// TwinCAT 3 PLC project MONETRuntime
// ProgramVersion: 3.1.4023.0
// libraries:
//   AstroBROT, * (BROT)
//   BROTLib, * (BROT)
//   Tc2_DataExchange, * (Beckhoff Automation GmbH)
//   Tc2_Math, * (Beckhoff Automation GmbH)
//   Tc2_MC2, * (Beckhoff Automation GmbH)
//   Tc2_MC2_Drive, * (Beckhoff Automation GmbH)
//   Tc2_NC, * (Beckhoff Automation GmbH)
//   Tc2_Standard, * (Beckhoff Automation GmbH)
//   Tc2_System, * (Beckhoff Automation GmbH)
//   Tc2_Utilities, * (Beckhoff Automation GmbH)
//   Tc3_IotBase, * (Beckhoff Automation GmbH)
//   Tc3_Module, * (Beckhoff Automation GmbH)
//   VisuDialogs, * (System)
//   VisuSymbols,3.5.10.0,System
// project tree:
//   DUTs/ E_Blink.TcDUT (not stored), E_Horn.TcDUT (not stored), E_TCSCommand.TcDUT (not stored), E_TCSErrors.TcDUT (not stored), E_TelescopeMode.TcDUT (not stored)
//   / GlobalTextList.TcGTLO, PlcTask.TcTTO (not stored), Visualization Manager.TcVMO (not stored)
//   GVLs/ GVL_Hydraulics.TcGVL (not stored), GVL_Main.TcGVL, GVL_pendant_control.TcGVL (not stored), GVL_Roof.TcGVL (not stored), GVL_Safety.TcGVL, GVL_Telescope.TcGVL
//   POUs/ AzimuthElevationControl.TcPOU, CoverControl.TcPOU, DerotatorControl.TcPOU, ElevationControl.TcPOU, FocusControl.TcPOU, HydraulicsControl.TcPOU, MAIN.TcPOU, PendantControl.TcPOU, RoofControl.TcPOU, PowerMonitoring.TcPOU, SafetyHandling.TcPOU, TelescopeAuxiliary.TcPOU, TelescopeControl.TcPOU
//   POUs/FunctionBlocks/ FB_AstroClock.TcPOU (not stored), FB_BLINK.TcPOU (not stored), FB_ButtonEnable.TcPOU (not stored), FB_Cover.TcPOU (not stored), FB_EventLog.TcPOU (not stored), FB_Horn.TcPOU (not stored), FB_LightTimer.TcPOU (not stored), FB_RFTRIG.TcPOU (not stored), FB_TimeAverage.TcPOU (not stored), FB_Timer.TcPOU (not stored), FB_TONTP.TcPOU (not stored), TelescopeAxisClass.TcPOU (not stored)
//   POUs/Functions/ CT2LST.TcPOU (not stored), F_Azimuthvelocity.TcPOU (not stored), F_DerotatorPosition2.TcPOU (not stored), F_Derotatorvelocity.TcPOU (not stored), F_Elevationvelocity.TcPOU (not stored), F_YREAL.TcPOU (not stored), NCError_TO_STRING.TcPOU (not stored), PointingModelAzimuth.TcPOU (not stored), PointingModelElevation.TcPOU (not stored), Refraction.TcPOU (not stored)
//   VISUs/ Hydraulics.TcVIS, Safety.TcVIS, Visualization.TcVIS

// ---- GVLs/GVL_Main.TcGVL
{attribute 'qualified_only'}
//TODO update to current RoboTel IOs
VAR_GLOBAL
	//DIN1 0.0
	//phase_available		AT%I*: BOOL;
	//not implemented on RoboTel
	//key_switch			AT%I*: BOOL;
	//DIN3 0.2
	key_switch_remote	AT%I*: BOOL;
	//DIN4 0.3
	start_switch		AT%I*: BOOL;
	//DIN5 0.4
	stop_switch			AT%I*: BOOL;
	//DIN8 0.7
	reset_switch		AT%I*: BOOL;
	
	//BT1
	main_cabinet_temperature	AT%I*: INT;
	//DIN15 1.6
	brake_clearing		AT%I*: BOOL;
	
	//DOUT1 0.0
	lamp_power			AT%Q*: BOOL;
	//DOUT2 0.1
	lamp_on_manual			AT%Q*: BOOL;
	//DOUT3 0.2
	lamp_error			AT%Q*: BOOL;
	
	(*
	NeutralCurrentGuardWarning		AT%I*:	BOOL;
	NeutralCurrentGuarError			AT%I*:	BOOL;
	ActivePowerGuardWarning			AT%I*:	BOOL;
	ActivePowerGuardError			AT%I*:	BOOL;
	ApparentPowerGuardWarning		AT%I*:	BOOL;
	ApparentPowerGuardError			AT%I*:	BOOL;
	*)
	//ActivePower						AT%I*:	REAL;
	//ActiveEnergy					AT%I*:	LINT;
	//NeutralLineCurrent				AT%I*:	REAL;
END_VAR

// ---- GVLs/GVL_Safety.TcGVL
{attribute 'qualified_only'}
VAR_GLOBAL
	// Safety Error Condition
	Error		AT%I*:	BOOL;
	// Run/Stop Safety
	Run			AT%Q*:	BOOL;
	// Restart Safety
	Restart		AT%Q*:	BOOL;
	// Error Acknowledgement 
	ErrAck		AT%Q*:	BOOL;
	// Stop signal coming from Safety
	// Stop		AT%I*:	BOOL;
	
	Reset_STO_Azimuth		AT%Q*: BOOL;
	Reset_STO_Elevation		AT%Q*: BOOL;
	Reset_STO_Derotator		AT%Q*: BOOL;
END_VAR

// ---- GVLs/GVL_Telescope.TcGVL
{attribute 'qualified_only'}
VAR_GLOBAL
	// DIN28 3.3 (absolute)
	azimut_limit_switch	AT%I*: BOOL;

	//Horn 4.7
	horn			AT%Q*: BOOL;
	
END_VAR

// ---- POUs/AzimuthElevationControl.TcPOU
PROGRAM AzimuthElevationControl
VAR_INPUT
	// enable the axis and its position control loop
	Enable:		BOOL;
	// reset the axis
	Reset: 		BOOL;
	// decrease azimuth
	left:		BOOL;
	// increase azimuth
	right: 		BOOL;
	// Move azimuth to given position
	MoveAxis:	BOOL;
	// Home the axis
	HomeAxis:	BOOL;
	// enable tracking
	Tracking:	BOOL;
	// position to move the axis to
	position: 	LREAL;
	// set the Velocity of the axis
	velocity:	LREAL;
	// stop the Axis
	StopAxis:	BOOL;
	// diagnostic reset
	bSoEReset:	BOOL;
	comm: I_Comm;
END_VAR
VAR_IN_OUT
	HydraulicsControl : FB_HydraulicsControl;
END_VAR
VAR_OUTPUT
	// error state of the axis
	error: 			BOOL;
	// error ID of the axis
	ErrorID:		UDINT;
	// actual_position of the axis
	act_position:	LREAL;
	// is the axis calibrated
	calibrated:		BOOL;
	// drive is ready
	ready:			BOOL;
	// time to reach target position
	slewtime:		LREAL;
END_VAR
VAR
	AzimuthAxis:		FB_Axis2;
	AzimuthCalibration: MC_SetPosition;
	//fbSoEReset:			FB_SoEReset;
	AzimuthAxisEvent: 	FB_EventLog;
	AzimuthDiagnosticEvent: 	FB_EventLog;
	// delay until commutator angle is measured
	readydelay:			TON;
	HomeDelay:			FB_TONTP;
	TorqueError:		TON := (PT := T#3S);
	azimuth_torque: 	REAL;
	TorqueWarning:		FB_EventLog;
	CalibrationEvent:	FB_Eventlog;
	ReadParameter:		MC_ReadParameter;
	getlastposition:	BOOL := TRUE;
	azimuth_rest_timer:	TON;
	azimuth_at_rest:	BOOL;
	fbSoEReset: 		FB_SoEReset;
	DiagnosticError:	BOOL;
END_VAR
VAR CONSTANT
	// reference position for homing
	// homing_position:		LREAL := 439.0; // was 442 - -21.21 = 463.21; 463 + 24 = 439
	// current position of the calibration cam encoder zero index. Apply an offset here if necessary
	calibration_position:	LREAL :=  212.75; //208.4983;//208.6273; //208.6073; // 208.7122869;//207.0092; // 208.2342; 
END_VAR
VAR PERSISTENT
	last_position:	LREAL := -1.0;
END_VAR

(* Azimuth Axis control section
Power must be on and brake must be open for the axis to operate
*)

// generate the ready signal after enabling the drive
readydelay(IN :=  AzimuthAxis.Enable, PT := T#3000MS, Q=> ready);

// limit the input position angle
position := LIMIT(0.0, position, 450.0);

// conduct the calibrated signal
calibrated := AzimuthAxis.Calibrated;

IF Calibrated OR Error THEN
	HomeAxis := FALSE;
	getlastposition := FALSE;
END_IF
	
IF HomeAxis THEN
	position := calibration_position;
END_IF

IF HomeDelay.Q THEN
	position := calibration_position;
	MoveAxis := TRUE;
END_IF

// perform a recalibration on the last known position
AzimuthCalibration(
	Axis := GVL_Telescope.AzimuthAxisRef,
	Execute := getlastposition AND last_position>=0.0 AND NOT Calibrated,
	Position := last_position);

IF AzimuthCalibration.Done THEN
	getlastposition := FALSE;
END_IF

IF Calibrated THEN
	last_position := act_position;
END_IF

// enable the azimuth if not moved by the power chain. Sorry for the hack
azimuth_rest_timer(IN := HydraulicsControl.brake_open AND 
				(ABS(GVL_Telescope.AzimuthAxisRef.NcToPlc.ActVelo) < 0.01), PT := T#2S);
// if azimuth at rest or calibrated, allow enabling the azimuth
IF azimuth_rest_timer.Q or calibrated THEN
	azimuth_at_rest := TRUE;
ELSIF HydraulicsControl.brake_closed THEN
	azimuth_at_rest := FALSE;
END_IF
	
// deactivate limit switches on homing
MC_SetAcceptBlockedDriveSignal(
	Axis := GVL_Telescope.AzimuthAxisRef, 
	Enable := HomeAxis);

AzimuthAxis(	
	Enable := 			enable AND azimuth_at_rest AND NOT GVL_Telescope.azimut_limit_switch,
	Reset := 			reset,
	MoveAxis :=			MoveAxis,
	HomeAxis := 		HomeAxis,
	StopAxis :=			StopAxis,
	Tracking :=			Tracking,
	Position := 		position, 
	Velocity :=			velocity,
	Enable_Positive := 	GVL_Telescope.Azimuth_inputs.1 OR HomeAxis,
	Enable_Negative := 	GVL_Telescope.Azimuth_inputs.0,
	Jog_Forward :=		right,
	Jog_Backwards := 	left,
	bCalibrationCam :=	NOT GVL_Telescope.Azimuth_inputs.1,
	ActualPosition => 	act_position,
	Error => 			error,
	ErrorID => 			ErrorID,
	AxisRef :=			GVL_Telescope.AzimuthAxisRef);

IF bSoEReset THEN
	last_position := -1.0;
	fbSoEReset(
		Axis := GVL_Telescope.AzimuthAxisRef,
		Execute := TRUE,
		Timeout := DEFAULT_ADS_TIMEOUT);
 	IF fbSoEReset.Busy THEN
		fbSoEReset(Axis := GVL_Telescope.AzimuthAxisRef, Execute := FALSE);
	ELSE
		bSoEReset := FALSE;
		Reset := TRUE;
	END_IF
END_IF 

IF AzimuthAxis.MoveDone THEN
	MoveAxis := FALSE;
END_IF

IF AzimuthAxis.HomeDone THEN
	HomeAxis := FALSE;
END_IF
	
IF AzimuthAxis.ResetDone THEN
	reset := FALSE;
END_IF

IF AzimuthAxis.StopDone THEN
	StopAxis := FALSE;
END_IF
DiagnosticError := FALSE;
IF GVL_Telescope.Azimuth_diagnostic < 16#D012 AND GVL_Telescope.Azimuth_diagnostic > 16#D014 THEN
	DiagnosticError :=TRUE;
	ErrorID := GVL_Telescope.Azimuth_diagnostic;
END_IF

ReadParameter(	Axis := GVL_Telescope.AzimuthAxisRef, Enable := AzimuthAxis.InMotion, 
				ParameterNumber := MC_AxisParameter.AxisRemainingTimeToGo, 
				ReadMode := E_ReadMode.READMODE_CYCLIC);
IF ReadParameter.Valid THEN
	slewtime := ReadParameter.Value;
END_IF

azimuth_torque := GVL_Telescope.Azimuth_torque / 10.0;
TorqueError(IN := ABS(azimuth_torque) > 50.0);


AzimuthAxisEvent(	
	Trigger := 		Error, 
	Level := 		ADSLOG_MSGTYPE_ERROR,
	FormatString :=	'Azimuth Axis Error: %s',
	OnMessage := 	NCError_TO_STRING(ErrorID),
	Comm := comm);
	
AzimuthDiagnosticEvent(	
	Trigger := 		DiagnosticError,
	Level := 		ADSLOG_MSGTYPE_ERROR,
	FormatString :=	'Azimuth Axis Diagnostic Error: %s',
	OnMessage := 	NCError_TO_STRING(GVL_Telescope.Azimuth_diagnostic),
	Comm := comm);
	
TorqueWarning(	
	Trigger := 		TorqueError.Q, 
	Level := 		ADSLOG_MSGTYPE_WARN,
	FormatString :=	'%s',
	OnMessage := 	'Azimuth torque is high.',
	Comm := comm);
	
CalibrationEvent(
	Trigger := 		Calibrated, 
	Level := 		ADSLOG_MSGTYPE_HINT,
	FormatString :=	'%s',
	OnMessage := 	'Azimuth axis is calibrated.',
	Comm := comm);

END_PROGRAM

// ---- POUs/HydraulicsControl.TcPOU
PROGRAM HydraulicsControl
VAR_INPUT
	// start the hydraulics
	enable:		BOOL := FALSE;
	// reset any hydraulics error
	reset: 		BOOL;
	// manual override to start the suction pump
	suction_manual:	BOOL;
	//manual override to stop the pump
	pump_manual_stop: BOOL;
END_VAR
VAR_OUTPUT
	// status of the brake: is the brake open?
	brake_open:			BOOL;
	// is the brake closed?
	brake_closed:		BOOL;
	// pump is running, but the pressure remains low
	pressure_failure:	BOOL;
	// suction was started, but it is not running
	suction_failure:	BOOL;
	// main pump is running but suction has a timeout
	hydraulics_failure:	BOOL;
	main_pump_failure: BOOL;
	// oil is low
	oil_low:			BOOL;
	// oil is high (unused?)
	oil_high:			BOOL;
	// oil pressure is 25 bars
	oil_pressure_OK:	BOOL;
	// oil is on reserve
	oil_warning:		BOOL;
	// oil filter is dirty
	oil_filter_dirty:	BOOL;
	// oil is below 10°C
	oil_cold:			BOOL;
	// oil is above 50°C
	oil_hot:			BOOL;
	// main pump is running
	pump_running:		BOOL;
	// suction pump is running
	suction_running :	BOOL := FALSE;
	// error condition
	error: 				BOOL;
END_VAR
VAR
	// command to open the brake
	iopen_brake:	BOOL := FALSE;
	// command to open the brake
	iclose_brake: BOOL;
	// monitors the pressure of the pump is running
	pressure_watchdog:	TON;
	// monitors the activation of the suction pump
	suction_watchdog: TON;
	// monitors the activation of the main pump
	main_pump_watchdog:	TON;
	// watch the hydraulics and suction pumps
	hydraulics_watchdog: TON;
	// represents the state of the main pump
	oil_pump_state:		RS;
	// represents the state of the brake
	brake_state: 		RS;
	// wait for the brake to open after pressure has been established
	brake_open_delay:	TON;
	// report brake opend after a short delay
	brake_opened_delay:	TON;
	// error state (set dominant)
	error_state:	SR;
	// trigger for suction pump
	suction_trigger:	SR;
	// timer to shut off hydraulics after break was closed
	hydraulics_off_timer:	TON  := (PT := T#300S);
	off_trigger:	F_TRIG;
	oil_level, last_oil_level:		REAL;
	HydraulicsLog,
	PumpLog,
	ReserveLog,
	oil_low_log,
	FilterLog,
	oil_max_log,
	OverTemperatureLog,
	UnderTemperatureLog,
	SuctionLog,
	HydraulicsFailureLog,
	BrakeClearingWarning,
	BrakeHydraulicsWarning,
	BrakeWarning: FB_EventLog;
	
	// measures the operating cycle of the suction pump
	StatusWord, LastStatus:	UDINT;
END_VAR

(* 
Main control Logic for the Hydraulics system
* power on delay for main pump and suction pump
* start main pump if main control is ready (button pressed or remote)
* start suction pump if maximum in pan is reached
* suction pump runs for 60 seconds
* stop main pump if oil is low
* stop main pump if pressure fails for 10 seconds
*)
oil_low := NOT GVL_Hydraulics.oil_low;
oil_high := NOT GVL_Hydraulics.oil_high;
oil_warning := GVL_Hydraulics.oil_reserve;
oil_pressure_OK := GVL_Hydraulics.oil_pressure_OK;
oil_filter_dirty := NOT GVL_Hydraulics.oilfilter_dirty;
oil_cold := NOT GVL_Hydraulics.oil_undertemperature;
oil_hot := GVL_Hydraulics.oil_overtemperature;
oil_level := F_YREAL(GVL_Hydraulics.oil_level, 0, 16383, 0.0, 5.0);
pump_running := GVL_Hydraulics.pump_running;
suction_running := GVL_Hydraulics.suction_running;

error_state(SET1 := pressure_failure OR	suction_failure OR hydraulics_failure OR oil_low OR main_pump_failure,
			RESET := reset,
			Q1 => error);
// clear reset, if no error present

IF NOT error THEN
	reset := FALSE;
END_IF

oil_pump_state(SET := enable,
				RESET1 := NOT enable OR error OR pump_manual_stop OR GVL_Hydraulics.oilpan_maximum);

GVL_Hydraulics.oil_pump_enable := oil_pump_state.Q1;

(* This section controls the hydraulic brake responsible for azimuth and elevation. 
Especially the elevation is imbalanced if not in the position control loop. 
The brake must only be opened, if the elevation drive is activated concurrently.
*)


// close the brake if the pump is not running	
IF iclose_brake OR NOT pump_running THEN 
	iopen_brake := FALSE;
END_IF

// wait for pressure to build up (hack for oil_pressure_ok)
brake_open_delay(IN := pump_running AND oil_pressure_OK,
				PT := T#3S);
		
brake_state(SET := brake_open_delay.Q AND iopen_brake AND MAIN.brake_clearing,
			RESET1 := GVL_Telescope.azimut_limit_switch 
					  OR iclose_brake 
					  OR NOT pump_running
					  OR NOT MAIN.brake_clearing,
			Q1 => GVL_Telescope.brake_azimuth_eve);

// signal that the brake is open after one second
brake_opened_delay(	IN :=brake_state.Q1, 
					PT := T#1000MS,
					Q => brake_open);

brake_closed := NOT brake_open;
IF brake_closed THEN
	iclose_brake := FALSE;
END_IF
// turn off the hydraulics if the brake is closed and the pump is still running
hydraulics_off_timer(IN := brake_closed AND enable );
off_trigger(CLK := hydraulics_off_timer.Q);

IF hydraulics_off_timer.Q THEN
	enable := FALSE;
END_IF

(* This is the end of the brake control section *)

suction_trigger(SET1 := GVL_Hydraulics.oilpan_maximum OR oil_level>2.9,
				RESET := oil_level<1.2);
GVL_Hydraulics.oil_suction_enable := suction_trigger.Q1 OR suction_manual;					
suction_watchdog(IN := GVL_Hydraulics.oil_suction_enable AND NOT suction_running,
					PT := T#15S,
					Q => suction_failure);
					
pressure_watchdog(IN := GVL_Hydraulics.oil_pump_enable AND 
						NOT oil_pressure_OK,
					PT := T#30S,
				  Q => pressure_failure);
hydraulics_watchdog(IN := pump_running AND NOT suction_running,
						PT := T#140S,
						Q => hydraulics_failure);

main_pump_watchdog(IN := GVL_Hydraulics.oil_pump_enable AND NOT pump_running,
					PT := T#10S,
					Q => main_pump_failure);

StatusWord.0 := oil_low;
StatusWord.1 := oil_high;
StatusWord.2 := oil_warning;
StatusWord.3 := oil_pressure_OK;
StatusWord.4 := oil_filter_dirty;
StatusWord.5 := oil_cold;
StatusWord.6 := oil_hot;
StatusWord.7 := brake_open;
StatusWord.8 := GVL_Main.brake_clearing;
StatusWord.9 := pump_running;
StatusWord.10 := suction_running;
StatusWord.11 := GVL_Hydraulics.oilpan_maximum;
StatusWord.12 := GVL_Hydraulics.oil_pump_enable;
StatusWord.13 := GVL_Hydraulics.oil_suction_enable;
IF ABS(last_oil_level - oil_level) > 0.02 THEN
	StatusWord.15 := TRUE;
	last_oil_level := oil_level;
ELSE
	StatusWord.15 := FALSE;
END_IF

IF StatusWord<>LastStatus THEN // publish new payload every second
	LastStatus := StatusWord;
	MAIN.MQTTClient.Publish('hydraulics', 'base', 'OilLow',			BOOL_TO_STRING(oil_low));
	MAIN.MQTTClient.Publish('hydraulics', 'base', 'OilHigh',		BOOL_TO_STRING(oil_high));
	MAIN.MQTTClient.Publish('hydraulics', 'base', 'OilMaximum',		BOOL_TO_STRING(GVL_Hydraulics.oilpan_maximum));
	MAIN.MQTTClient.Publish('hydraulics', 'base', 'OilReserve',		BOOL_TO_STRING(oil_warning));
	MAIN.MQTTClient.Publish('hydraulics', 'base', 'OilPressureOK', 	BOOL_TO_STRING(oil_pressure_OK));
	MAIN.MQTTClient.Publish('hydraulics', 'base', 'OilFilterDirty',	BOOL_TO_STRING(oil_filter_dirty));
	MAIN.MQTTClient.Publish('hydraulics', 'base', 'OilCold',		BOOL_TO_STRING(oil_cold));
	MAIN.MQTTClient.Publish('hydraulics', 'base', 'OilHot',			BOOL_TO_STRING(oil_Hot));
	MAIN.MQTTClient.Publish('hydraulics', 'base', 'BrakeOpen',		BOOL_TO_STRING(brake_open));
	MAIN.MQTTClient.Publish('hydraulics', 'base', 'BrakeClearing',	BOOL_TO_STRING(GVL_Main.brake_clearing));
	MAIN.MQTTClient.Publish('hydraulics', 'base', 'PumpRunning',	BOOL_TO_STRING(pump_running));
	MAIN.MQTTClient.Publish('hydraulics', 'base', 'SuctionRunning',	BOOL_TO_STRING(suction_running));
	MAIN.MQTTClient.Publish('hydraulics', 'base', 'OilLevel',		REAL_TO_STRING(oil_level));
	MAIN.MQTTClient.Publish('hydraulics', 'base', 'StatusWord',		UDINT_TO_STRING(StatusWord));
END_IF


				  				  
HydraulicsLog(Trigger := pressure_failure OR main_pump_failure,
				Level := ADSLOG_MSGTYPE_ERROR,
				FormatString := 'Main hydraulics pump / pressure: %s',
				OnMessage := 'FAILURE',
				OffMessage := 'OK',
				OffLevel := ADSLOG_MSGTYPE_HINT);

PumpLog(Trigger := pump_running,
				Level := ADSLOG_MSGTYPE_HINT,
				FormatString := 'Main hydraulics pump: %s',
				OnMessage := 'START',
				OffMessage := 'STOP',
				OffLevel := ADSLOG_MSGTYPE_HINT);
	
ReserveLog(Trigger := oil_warning,
			Level := ADSLOG_MSGTYPE_WARN,
			FormatString := 'oil reserve: %s',
			OnMessage := 'LOW',
			OffMessage := 'OK',
			OffLevel := ADSLOG_MSGTYPE_HINT);

oil_low_log(Trigger := oil_low,
				Level := ADSLOG_MSGTYPE_ERROR,
				FormatString := 'oil level: %s',
				OnMessage := 'LOW',
				OffMessage := 'OK',
				OffLevel := ADSLOG_MSGTYPE_HINT);

oil_max_log(Trigger := GVL_Hydraulics.oilpan_maximum,
				Level := ADSLOG_MSGTYPE_ERROR,
				FormatString := 'oil level: %s',
				OnMessage := 'MAXIMUM',
				OffMessage := 'OK',
				OffLevel := ADSLOG_MSGTYPE_HINT);	
				
FilterLog(Trigger := oil_filter_dirty,
				Level := ADSLOG_MSGTYPE_WARN,
				FormatString := 'Hydraulics Filter is %s',
				OnMessage := 'dirty.');

OverTemperatureLog(Trigger := oil_hot,
				Level := ADSLOG_MSGTYPE_WARN,
				FormatString := 'Hydraulics Temperature is %s',
				OnMessage := 'high.');
				
UnderTemperatureLog(Trigger := oil_cold,
				Level := ADSLOG_MSGTYPE_WARN,
				FormatString := 'Hydraulics Temperature is %s',
				OnMessage := 'low.');

SuctionLog(Trigger := suction_failure,
				Level := ADSLOG_MSGTYPE_ERROR,
				FormatString := 'suction pump: %s',
				OnMessage := 'FAILURE',
				OffMessage := 'OK',
				OffLevel := ADSLOG_MSGTYPE_HINT);

HydraulicsFailureLog(Trigger := hydraulics_failure,
				Level := ADSLOG_MSGTYPE_ERROR,
				FormatString := 'suction pump while running main pump: %s',
				OnMessage := 'FAILURE',
				OffMessage := 'OK',
				OffLevel := ADSLOG_MSGTYPE_HINT);
				
BrakeClearingWarning(Trigger := NOT Main.brake_clearing AND iopen_brake,
				Level := ADSLOG_MSGTYPE_WARN,
				FormatString := '%s',
				OnMessage := 'Cannot open brake without brake clearing.');

BrakeWarning(	Trigger := brake_open,
				Level := ADSLOG_MSGTYPE_WARN,
				FormatString := '%s',
				OnMessage := 'Brake is open.',
				OffMessage := 'Brake is closed.');

BrakeHydraulicsWarning(Trigger := NOT enable AND iopen_brake,
				Level := ADSLOG_MSGTYPE_WARN,
				FormatString := '%s',
				OnMessage := 'Cannot open brake without running hydraulics.');

METHOD close_brake : BOOL
VAR_INPUT
END_VAR
// close the brake
iclose_brake := TRUE;

RETURN(brake_closed);
END_METHOD

METHOD open_brake : BOOL
VAR_INPUT
END_VAR
// start the pump
enable := TRUE;
// open the brake
IF oil_pressure_OK THEN
	iopen_brake := TRUE;
END_IF;
RETURN(brake_open);
END_METHOD

END_PROGRAM

// ---- POUs/MAIN.TcPOU
PROGRAM MAIN
VAR
	ready				: BOOL;		// telescope drives are ready to enable
	error				: BOOL;		// error stat on drive, power or hydraulics
	brakeClearing		: BOOL := FALSE;	//	open brake
	
	commTimer 			: TON := (PT:=T#5S);
	getHostName			: FB_GetHostName;
	hostName			: STRING(255);
	executeHostName		: BOOL := TRUE;
	
	eTelescopeMode 		: E_TelescopeMode;
	
	fbComm				: FB_Comm_MQTT_Influx;
	SafetyHandling		: FB_MonetSafetyHandling(comm := fbComm);
	CabinetControl		: FB_MonetCabinetControl(comm := fbComm);
	PowerMonitoring		: FB_MonetPowerMonitoring(comm := fbComm);
	RoofControl			: FB_RoofControl(comm := fbComm);
	CoverControl		: FB_MonetCoverControl(comm := fbComm);
	HydraulicsControl	: FB_HydraulicsControl(comm := fbComm);
	FocusControl		: FB_FocusControl(comm := fbComm);
	DerotatorControl	: FB_DerotatorControl(comm := fbComm);
	ElevationControl	: FB_ElevationControl(comm := fbComm);
	AzimuthControl		: FB_AzimuthControl(comm := fbComm);
	TelescopeControl	: FB_MonetTelescopeControl(comm := fbComm);
	PendantControl		: FB_MonetPendantControl(comm := fbComm);
	MqttWatchdog		: FB_MonetMqttWatchdog(comm := fbComm);	// park + close roof after 30 s without broker (MONETcommon)
	Diagnostics			: FB_MonetDiagnostics(comm := fbComm);	// diagnostics/base/* telemetry, on change + 30 s heartbeat (MONETcommon)
END_VAR
VAR CONSTANT
	telescopeConfig		: ST_TelescopeConfig := (longitude := -104.0217, latitude := 30.6714, altitude := 2000.0, 
												 azimuthPark := 190, elevationPark := 60, derotatorPark := -116.42, focusPark := 53.8, 
												 azimuthHome := 190, elevationHome := 40, derotatorHome := -116.42,
												 name := 'MONET/N', diameter := 1.2, cabinet := 'Beckhoff', manufacturer := 'Halfmann, Haidenhain, Beckhoff',
												 mountOptions := 'ALT-AZ', mount := 'ALT_AZ');
	// MONET/N pointing model, moved here from its former local copy of FB_MonetTelescopeControl (same coefficients)
	fbPointing			: FB_PointingModelForward(AOFF := 0.0, BNP := 0.41799581014823517, AN_A := -0.0005399238415356825, AE_A := 0.0010943700155200701, NPAE := 0.3540915955287274,
                                                  EOFF := 0.0, AN_E := -0.0015387935505830619, AE_E := 0.0028384915610841777, TF := 0.07539398326327973);
	fbPointingInverse	: FB_PointingModelInversion(fbPointing := fbPointing);
END_VAR

(* 
Main control loop
* Execute sub modules
* power management
* control panel switches and status lamps

* start switch activates Hydraulics and Trafo
* 
*)

// get hostname for MQTT connection
GetHostName(bExecute := executeHostName, sHostName => HostName);
executeHostName := FALSE;

// run cabinet
CabinetControl();

// telescope mode
IF CabinetControl.KeyLocal THEN
	eTelescopeMode := SEL(HydraulicsControl.Enable, E_TelescopeMode.off, E_TelescopeMode.manual);	
ELSE
	eTelescopeMode := E_TelescopeMode.automatic; 
END_IF

// in local mode we can start or stop hydraulics and open the brake
brakeClearing := TRUE;
IF eTelescopeMode = E_TelescopeMode.manual OR eTelescopeMode = E_TelescopeMode.off THEN
	IF CabinetControl.IsStartPushed() THEN
		HydraulicsControl.Enable := TRUE;
	END_IF
	IF CabinetControl.IsStopPushed() THEN
		HydraulicsControl.Enable := FALSE;
	END_IF
	brakeClearing := CabinetControl.AreBreakesCleared();
	HydraulicsControl.bOpenBrake := brakeClearing;
END_IF

// clear errors: SafetyHandling.resetRequest (see call below) toggles Restart/ErrAck,
// here the cabinet/pendant reset button also resets covers, hydraulics and, in automatic mode, the
// telescope control (the only way to clear a latched bInterrupted)
IF CabinetControl.IsResetPushed() OR PendantControl.IbResetButton THEN
	CoverControl.Reset();
	HydraulicsControl.Reset();
	IF eTelescopeMode = E_TelescopeMode.automatic THEN
		TelescopeControl.Reset();
	END_IF
END_IF

// telescope is ready when power available
PowerMonitoring(phaseOK => ready);

// only run TelescopeControl in automatic mode
IF eTelescopeMode = E_TelescopeMode.automatic THEN
	TelescopeControl(
		telescopeConfig := telescopeConfig,
		fbCovers 		:= CoverControl,
		fbBrake 		:= HydraulicsControl,
		fbHydraulics 	:= HydraulicsControl,
		fbFocus 		:= FocusControl,
		fbElevation 	:= ElevationControl,
		fbAzimuth 		:= AzimuthControl,
		fbDerotator 	:= DerotatorControl,
		fbPointing      := fbPointing,
		fbPointingInverse := fbPointingInverse,
		bEstopTriggered := SafetyHandling.estop,	// M5: was never wired, see MONETcommon#11
		bMainReady		:= ready					// M5: was computed and published but never wired, see MONETcommon#11
	);
END_IF

// run all control FBs
CoverControl();
HydraulicsControl(
	nMinPanLevel	:= 3000,
	nMaxPanLevel	:= 10200,
	fMinPanPercent	:= 0.0,
	fMaxPanPercent	:= 50.0, //56.0,
	bBrakeClearing	:= brakeClearing
);
ElevationControl(
	fCalibPosition 	:= 25.8657627917962052,
	fbCovers 		:= CoverControl, 
	fbBrake 		:= HydraulicsControl
);
AzimuthControl(
	fCalibPosition	:=  211.355503610763347,
	fMinPosition	:= -72.0,
	fMaxPosition	:= 495.0,
	bBrakeOpen		:= HydraulicsControl.brakeOpen,
);
DerotatorControl(
	fMinPosition		:= -170.0,
	fMaxPosition		:= 300.0
);	//
FocusControl(
	eTelescopeMode 	:= eTelescopeMode,
	fHomingPosition	:= 92.02, // 104.02 - 12.00
	fVelocity		:= 0.2
);
RoofControl(
	min_speed		:= 10000,
	max_speed 		:= 30000, 
	acceleration 	:= 150,
	min_position_1 	:= 0,
	max_position_1 	:= 202,
	min_position_2 	:= 0,
	max_position_2 	:= 202,
	max_position_diff	:= 3,
	limit_slowdown	:= 5
);
PendantControl(
	fbCovers 		:= CoverControl, 
	fbBrake 		:= HydraulicsControl, 
	fbHydraulics 	:= HydraulicsControl, 
	fbFocus 		:= FocusControl, 
	fbElevation 	:= ElevationControl, 
	fbAzimuth 		:= AzimuthControl, 
	fbDerotator 	:= DerotatorControl	
);

// broker gone for 30 s: park the telescope and close the roof (armed after the first connect)
MqttWatchdog(bConnected := fbComm.bConnected, iTelescope := TelescopeControl, iRoof := RoofControl);

// and fbComm
fbComm(
	sHostName		:= '169.254.146.10',
    nHostPort  		:= 1883,
    nKeepAlive  	:= 60,
	sTopicSub  		:= 'MONETN/Telescope/SET',
	sTopicPublish	:= 'MONETN/Telemetry',
	sTopicLog		:= 'MONETN/Log',
	Telescope		:= TelescopeControl,
	AltAzTelescope  := TelescopeControl,
	Focus			:= FocusControl,
	Roof			:= RoofControl
);

// set control lights
//error := Focuscontrol.Error OR CoverControl.Error OR HydraulicsControl.Error;
error := CoverControl.Error OR HydraulicsControl.Error;
CabinetControl.SetManualLamp(eTelescopeMode = E_TelescopeMode.manual);

// blink errors
IF SafetyHandling.error THEN
	CabinetControl.SetBlinkError(E_Blink.short);
ELSIF ElevationControl.bError OR AzimuthControl.bError OR DerotatorControl.bError THEN
	CabinetControl.SetBlinkError(E_Blink.long);
ELSIF HydraulicsControl.bOilWarning OR HydraulicsControl.bOilHot OR HydraulicsControl.bPressureFailure THEN
	CabinetControl.SetBlinkError(E_Blink.slow);
ELSIF error THEN
	CabinetControl.SetBlinkError(E_Blink.on);
ELSE
	CabinetControl.SetBlinkError(E_Blink.off); 
END_IF

// power lamp is always on
CabinetControl.SetBlinkPower(E_Blink.on);

// do safety
SafetyHandling(resetRequest := CabinetControl.IsResetPushed() OR PendantControl.IbResetButton);

// telemetry
commTimer(IN:=TRUE);
IF commTimer.Q THEN
	commTimer(IN:=FALSE);
	fbComm.Publish('electronics', 'base', 'MainReady', BOOL_TO_STRING(ready));
	fbComm.Publish('electronics', 'base', 'MasterError', BOOL_TO_STRING(error));
END_IF

// diagnostics telemetry: publish on change, plus a full-snapshot heartbeat (MONETcommon)
Diagnostics(
	fbTelescope	:= TelescopeControl,
	fbElevation	:= ElevationControl,
	fbAzimuth	:= AzimuthControl,
	fbDerotator	:= DerotatorControl,
	fbFocus		:= FocusControl,
	fbSafety	:= SafetyHandling
);

END_PROGRAM

// ---- POUs/SafetyHandling.TcPOU
PROGRAM SafetyHandling
VAR
	state           : INT := 0;            
	// power on delay
	start_delay 	: TON := (PT := T#2S);
	state_delay 	: TON := (PT := T#1S);

	// Safety group
	fbInfoGroup1			:FB_InfoGroup;
	stInfoGroup1	AT%I*	:ST_InfoDataGroup;
	sStateGroup1			:STRING;
	
	// Estop
	fbInfoEStop1			:FB_InfoEStop;
	stInfoEStop1 	AT%I*	:ST_InfoDataFB;
	sStateEStop1			:STRING;
	sDiagEStop1				:STRING;	
	
	// Info EL1904
	fbInfoSafetyIn			:FB_InfoConnection;
	stInfoSafetyIn 	AT%I*	:ST_InfoDataConnection;
	sStateSafetyIn			:STRING;
	sDiagSafetyIn			:STRING;
	bSafetyInCh1			:BOOL;
	bSafetyInCh2			:BOOL;
	bSafetyInCh3			:BOOL;
	bSafetyInCh4			:BOOL;
	
	// Info EL2904
	fbInfoSafetyOut			:FB_InfoConnection;
	stInfoSafetyOut AT%I*	:ST_InfoDataConnection;
	sStateSafetyOut			:STRING;
	sDiagSafetyOut			:STRING;
	bSafetyOutCh1			:BOOL;
	bSafetyOutCh2			:BOOL;
	bSafetyOutCh3			:BOOL;
	bSafetyOutCh4			:BOOL;
	
	// Errack logging
	ErrAckLog		: FB_EventLog;
	// restart logging
	RestartLog		: FB_EventLog;
	// safety logging
	SafetyLog		: FB_EventLog;
	
END_VAR
VAR_OUTPUT
	// error condition
	Error			: BOOL;
	// Emergency_stop engaged
	Emergency_stop	: BOOL;
END_VAR
VAR_INPUT
	// issue a remote restart
	remote_restart:		BOOL;
	// issue a remute run/stop
	remote_run:			BOOL := TRUE;
END_VAR

// Safety is running on start
GVL_Safety.Run := remote_run;

fbInfoGroup1(
	stInfoData	:= stInfoGroup1,
	sState		=> sStateGroup1);

fbInfoEStop1(
	stInfoData	:= stInfoEStop1, 
	sState		=> sStateEStop1, 
	sDiag		=> sDiagEStop1);

//Info SafetyIn EL1904
fbInfoSafetyIn(
	stInfoData		:=stInfoSafetyIn, 
	sState			=>sStateSafetyIn, 
	sDiag			=>sDiagSafetyIn, 
	bChannel1		=>bSafetyInCh1, 
	bChannel2		=>bSafetyInCh2, 
	bChannel3		=>bSafetyInCh3, 
	bChannel4		=>bSafetyInCh4);	
	
//Info SafetyOut EL2904
fbInfoSafetyOut(
	stInfoData		:=stInfoSafetyOut, 
	sState			=>sStateSafetyOut, 
	sDiag			=>sDiagSafetyOut, 
	bChannel1		=>bSafetyOutCh1, 
	bChannel2		=>bSafetyOutCh2, 
	bChannel3		=>bSafetyOutCh3, 
	bChannel4		=>bSafetyOutCh4);
	
(*

// power on delay for Safety RESTART after RUN=1
start_delay(IN := TRUE);

CASE state OF
	0:
	    IF start_delay.Q  THEN
			GVL_Safety.ErrAck := TRUE;
			state := 1;
		END_IF
	1:
		state_delay(IN := TRUE);	
		IF state_delay.Q THEN
			GVL_Safety.ErrAck := FALSE;
			GVL_Safety.Restart := TRUE;
			state := 2;
			state_delay(IN := FALSE);
		END_IF
	2:
		state_delay(IN := TRUE);	
		IF state_delay.Q THEN
			GVL_Safety.Restart := FALSE;
			GVL_Safety.ErrAck := TRUE;
			state := 3;
			state_delay(IN := FALSE);
		END_IF
	3:
		state_delay(IN := TRUE);	
		IF state_delay.Q THEN	
			GVL_Safety.ErrAck := FALSE;
			state := 4;
			state_delay(IN := FALSE);
		END_IF	
END_CASE

// remote restart
IF remote_restart THEN
	state := 0;
	remote_restart := FALSE;
END_IF

// manual Err_Ack 
GVL_Safety.ErrAck := (GVL_Main.key_switch_remote AND GVL_Main.reset_switch);

// manual Restart
GVL_Safety.Restart := (GVL_Main.key_switch_remote AND GVL_Main.start_switch);

ErrAckLog(	Trigger := GVL_Safety.ErrAck,
			OnMessage := 'Safety error was acknowledged.');
			
RestartLog(	Trigger := GVL_Safety.Restart,
			Level := ADSLOG_MSGTYPE_WARN,
			OnMessage := 'Safety was restarted.');

SafetyLog(	Trigger := Error,
			Level := ADSLOG_MSGTYPE_ERROR,
			OnMessage := 'Safety Error! Emergency stop enganged!',
			OffMessage := 'Safety is OK.',
			OffLevel := ADSLOG_MSGTYPE_HINT);
*)

(*
// wait n seconds after Start ...
start_delay(IN := TRUE);
// ... and send ErrAck for n milliseconds
ErrAck_Pulse(IN := (GVL_Safety.State = 2) AND start_delay.Q);

// Error Acknowledgment: Turn key_switch OFF and press STOP 
GVL_Safety.ErrAck := (GVL_Main.key_switch_remote AND GVL_Main.reset_switch)
					OR ErrAck_Pulse.Q
					OR remote_ErrAck;
// detect falling edge 
ErrAck_Trigger(CLK := GVL_Safety.ErrAck);
// send restart pulse on falling edge of ErrAck
restart_pulse(IN := ErrAck_Trigger.Q);

// RESTART Safety after pushing reset or power on delay
GVL_Safety.Restart := (GVL_Main.key_switch_remote AND GVL_Main.start_switch)
 					   OR remote_restart
                       OR restart_pulse.Q;
				
//Error := GVL_Safety.Error OR (GVL_Safety.State <> 1);

//Emergency_stop := NOT GVL_Safety.Stop;

ErrAckLog(	Trigger := GVL_Safety.ErrAck,
			OnMessage := 'Safety error was acknowledged.');
			
RestartLog(	Trigger := GVL_Safety.Restart,
			Level := ADSLOG_MSGTYPE_WARN,
			OnMessage := 'Safety was restarted.');

SafetyLog(	Trigger := Error,
			Level := ADSLOG_MSGTYPE_ERROR,
			OnMessage := 'Safety Error! Emergency stop enganged!',
			OffMessage := 'Safety is OK.',
			OffLevel := ADSLOG_MSGTYPE_HINT);
*)

END_PROGRAM

// ---- POUs/PowerMonitoring.TcPOU
PROGRAM PowerMonitoring
VAR_INPUT
	comm: I_Comm;
END_VAR
VAR_OUTPUT
	phaseOK:				BOOL;
END_VAR
VAR
	Overvoltage				AT%I*: BOOL;
	Overcurrent				AT%I*: BOOL;
	VoltageGuardWarning		AT%I*: BOOL;
	VoltageGuardError		AT%I*: BOOL;
	CurrentGuardWarning		AT%I*: BOOL;
	CurrentGuardError		AT%I*: BOOL;
	Voltage					AT%I*: REAL;
	Current					AT%I*: REAL;
	ActivePower				AT%I*: REAL;
	ApparentPower			AT%I*: REAL;
	ReactivePower			AT%I*: REAL;
	PowerQualityFactor		AT%I*: REAL;
	Frequency				AT%I*: REAL;
	PowerFactor				AT%I*: REAL;
	NeutralLineCurrent		AT%I*: REAL;
	L1L2Voltage				AT%I*: REAL;
	L2L3Voltage				AT%I*: REAL;
	L3L1Voltage				AT%I*: REAL;
	MQTTTimer: 				TON := (PT:=T#10S);
	PowerWarningDelay:		TON := (PT:=T#100MS);
	PowerWarningRetain:		TOF := (PT:=T#2000MS);
	
	PowerError:				FB_EventLog;
	PowerWarning:			FB_EventLog;
	NeutralCurrentEvent:			FB_EventLog;
END_VAR

phaseOK := L1L2Voltage > 360.0 AND L2L3Voltage > 360.0 AND L3L1Voltage > 360.0;

IF NeutralLineCurrent > 0.1 THEN
	NeutralCurrentEvent.Trigger := TRUE;
	NeutralCurrentEvent.OnMessage := 	'Neutral Line Current WARNING!';
	NeutralCurrentEvent.Level := ADSLOG_MSGTYPE_WARN;
ELSIF NeutralLineCurrent > 0.3 THEN
	NeutralCurrentEvent.Trigger := TRUE;
	NeutralCurrentEvent.OnMessage := 	'Neutral Line Current ERROR!';
	NeutralCurrentEvent.Level := ADSLOG_MSGTYPE_ERROR;
ELSE
	NeutralCurrentEvent.Trigger := FALSE;
END_IF

PowerWarningDelay(IN := VoltageGuardWarning OR CurrentGuardWarning);
PowerWarningRetain(IN := PowerWarningDelay.Q);

// MQTT Section
MQTTTimer(IN:=TRUE);
IF MQTTTimer.Q OR VoltageGuardWarning OR CurrentGuardWarning THEN // publish new payload every second
	MQTTTimer(IN:=FALSE);

	comm.Publish('telescope', 'power', 'Overvoltege',	BOOL_TO_STRING(Overvoltage));
	comm.Publish('telescope', 'power', 'Overcurrent',	BOOL_TO_STRING(Overcurrent));

	comm.Publish('telescope', 'power', 'VoltageGuardWarning',	BOOL_TO_STRING(VoltageGuardWarning));
	comm.Publish('telescope', 'power', 'VoltageGuardError',		BOOL_TO_STRING(VoltageGuardError));
	comm.Publish('telescope', 'power', 'CurrentGuardWarning',	BOOL_TO_STRING(CurrentGuardWarning));
	comm.Publish('telescope', 'power', 'CurrentGuardError',		BOOL_TO_STRING(CurrentGuardError));

	comm.Publish('telescope', 'power', 'Voltage', 		REAL_TO_STRING(Voltage));
	comm.Publish('telescope', 'power', 'Current',		REAL_TO_STRING(Current));
	comm.Publish('telescope', 'power', 'ActivePower',	REAL_TO_STRING(ActivePower));
	comm.Publish('telescope', 'power', 'ApparentPower',	REAL_TO_STRING(ApparentPower));
	comm.Publish('telescope', 'power', 'ReactivePower',	REAL_TO_STRING(ReactivePower));
	comm.Publish('telescope', 'power', 'PowerQualityFactor',	REAL_TO_STRING(PowerQualityFactor));
	comm.Publish('telescope', 'power', 'Frequency',		REAL_TO_STRING(Frequency));
	comm.Publish('telescope', 'power', 'PowerFactor',	REAL_TO_STRING(PowerFactor));
	comm.Publish('telescope', 'power', 'NeutralLineCurrent',	REAL_TO_STRING(NeutralLineCurrent));

	comm.Publish('telescope', 'power', 'L1L2Voltage',	REAL_TO_STRING(L1L2Voltage));
	comm.Publish('telescope', 'power', 'L2L3Voltage',	REAL_TO_STRING(L2L3Voltage));
	comm.Publish('telescope', 'power', 'L3L1Voltage',	REAL_TO_STRING(L3L1Voltage));	
END_IF

// EventLog section
PowerError(	
	Trigger := 		VoltageGuardError OR CurrentGuardError, 
	Level := 		ADSLOG_MSGTYPE_ERROR,
	FormatString :=	'%s',
	OnMessage := 	'electrical power:	ERROR!');
	
PowerWarning(	
	Trigger := 		PowerWarningRetain.Q, 
	Level := 		ADSLOG_MSGTYPE_WARN,
	FormatString :=	'%s',
	OnMessage := 	'electrical power:	WARNING!');

NeutralCurrentEvent(
	FormatString :=	'%s',
	OnMessage := 	'electrical power:	WARNING!');

END_PROGRAM

// ---- POUs/RoofControl.TcPOU
PROGRAM RoofControl
VAR CONSTANT
	// max speed
	MAX_SPEED					: LREAL := 1;
END_VAR
VAR
	// commands for roofs
	open_roof1					: BOOL;
	close_roof1					: BOOL;
	stop_roof1					: BOOL;	
	open_roof2					: BOOL;
	close_roof2					: BOOL;
	stop_roof2					: BOOL;
	
	// open/closed status signals for both roofs (2 each)
	roof_open			AT%I*	: ARRAY[1..4] OF BOOL;
	roof_closed			AT%I*	: ARRAY[1..4] OF BOOL;
	
	// move direction for both roofs (2 each)
	roof_direction		AT%Q*	: ARRAY[1..4] OF BOOL;
	
	// move speed for both roofs (2 each)
	roof_moving					: ARRAY[1..4] OF BOOL;
	roof_vel_ramp				: ARRAY[1..4] OF FB_CTRL_RAMP_GENERATOR;
	roof_speed			AT%Q*	: ARRAY[1..4] OF LREAL;
	roof_target_speed	AT%Q*	: ARRAY[1..4] OF LREAL;	
	
	// ramp parameters for starting movement
	ramp_params			: ST_CTRL_RAMP_GENERATOR_PARAMS := (fVeloPos := 1, fVeloNeg := 1, tTaskCycleTime := T#100MS, tCtrlCycleTime := T#100MS);
	
	// loop variable	
	i					: INT;
END_VAR

// commands
IF open_roof1 THEN
	open_roof(1);
	open_roof1 := FALSE;
END_IF
IF open_roof2 THEN
	open_roof(2);
	open_roof2 := FALSE;
END_IF

// velocity ramps
FOR i := 1 TO 4 BY 1 DO
	roof_vel_ramp[i](
		bEnable		:= roof_moving[i],
		fStart		:= roof_speed[i],
		fTarget		:= roof_target_speed[i],
		stParams	:= ramp_params,
		fOut		=> roof_speed[i]);
END_FOR;
	
// stop on limit switches
FOR i := 1 TO 4 BY 1 DO
    IF roof_open[i] OR roof_closed[i] OR NOT roof_moving[i] THEN
		stop_motor(i);
	END_IF
END_FOR;

METHOD open_roof : BOOL
VAR_INPUT
	roof: INT;
END_VAR
VAR
	i: INT;	
END_VAR
FOR i := 0 TO 1 BY 1 DO
	roof_moving[2*(roof-1) + i] := TRUE;
	roof_direction[2*(roof-1) + i] := TRUE;
	roof_target_speed[2*(roof-1) + i] := MAX_SPEED;
END_FOR;
END_METHOD

METHOD stop_motor : BOOL
VAR_INPUT
	roof: INT;
END_VAR
roof_speed[roof] := 0;
roof_moving[roof] := FALSE;
END_METHOD

END_PROGRAM

// ---- POUs/CoverControl.TcPOU
PROGRAM CoverControl
VAR_INPUT
	// resets all drives after an error has occured
	reset:		BOOL;
	// open the cover in proper order
	open:		BOOL;
	// close the cover in proper order
	close:		BOOL;
	// actual active cover in manual mode, 0 for automatic = all covers active
	active_cover:	INT;

END_VAR
VAR_OUTPUT
	// is TRUE, if all covers are open
	isopen:			BOOL;
	// is TRUE, if all covers are closed
	isclosed:		BOOL;
	// is TRUE if any cover-driver reports an error
	Error: 	BOOL;
	// warning state of the DC drives
	Warning: BOOL;
	// cover1 is open
	Cover1_opened, 
	// cover1 is closed
	Cover1_closed:	BOOL;
	// cover2 is open
	Cover2_opened, 
	// cover2 is closed
	Cover2_closed:	BOOL;
	// cover3 is open
	Cover3_opened, 
	// cover3 is closed
	Cover3_closed:	BOOL;
	Cover1_error: BOOL;
	Cover2_error: BOOL;
	Cover3_error: BOOL;
END_VAR
VAR
	// delay timer for opening cover2
	open2_delay: 	TON := (PT:=T#1S);;
	// dely timer for closing cover3
	close3_delay : 	TON := (PT:=T#3S);;
	// trigger for error
	error_trigger:	SR;
	//error event for cover1
	Cover1_Event,
	Cover2_Event,
	Cover3_Event:	FB_EventLog;
	// timeout event for cover1
	Cover1_Timeout_Event,
	Cover2_Timeout_Event,
	Cover3_Timeout_Event:	FB_EventLog;
	// log if covers are open
	Covers_opened_event,
	// log if covers are closed
	Covers_closed_event:	FB_EventLog;
	// Event log for a generic drive error
	Covers_Error_event:		FB_EventLog;
	// Event log for a generic drive warning
	Covers_Warning_event:		FB_EventLog;
END_VAR

(*
This is the control for the two (three) telescope covers. 
The correct order for opening is 1->3->2 and for closing 2->3->1.
GVL Open and close signals are inverted
*)

// close has precedence over open
IF close THEN
	open := FALSE;
END_IF

Cover1_opened := NOT GVL_Telescope.cover1_open;
Cover2_opened := NOT GVL_Telescope.cover2_open;
Cover3_opened := NOT GVL_Telescope.cover3_open;
Cover1_closed := NOT GVL_Telescope.cover1_closed;
Cover2_closed := NOT GVL_Telescope.cover2_closed;
Cover3_closed := NOT GVL_Telescope.cover3_closed;
Cover1_error := Cover1_opened AND Cover1_closed;
Cover2_error := Cover2_opened AND Cover2_closed;
Cover3_error := Cover3_opened AND Cover3_closed;

// wait for cover2 until cover3 has left the closed state
open2_delay(IN := open AND NOT cover3_closed);
// wait for cover3 until cover2 has left the open state
close3_delay(IN := close AND NOT cover2_opened);

IF close THEN
	GVL_Telescope.close_cover1 := GVL_Telescope.cover1_closed AND NOT GVL_Telescope.cover3_closed;
	GVL_Telescope.close_cover2 := GVL_Telescope.cover2_closed;
	GVL_Telescope.close_cover3 := GVL_Telescope.cover3_closed AND close3_delay.Q;
ELSIF open THEN
	GVL_Telescope.open_cover1 := GVL_Telescope.cover1_open;
	GVL_Telescope.open_cover2 := GVL_Telescope.cover2_open AND open2_delay.Q;
	GVL_Telescope.open_cover3 := GVL_Telescope.cover3_open;			
END_IF


// we are open, if all covers are open
isopen := cover3_opened AND cover2_opened AND cover1_opened;
// we are closed, if all covers are closed
isclosed := cover2_closed AND cover3_closed AND cover1_closed;
// error indicates an axis error on any axis
error_trigger(SET1 := Cover1_error OR Cover2_error OR Cover3_error,
				RESET := reset,
				Q1 => error);
//Warning := Cover1_control.Warning OR Cover2_control.Warning OR Cover3_control.Warning;

IF isclosed THEN
	close := FALSE;
END_IF

IF isopen THEN
	open := FALSE;
END_IF

Covers_Error_Event.OnMessage := 'Cover drive error';
IF Error THEN
	IF Cover3_error THEN 
		Covers_Error_Event.OnMessage := 'Cover 3 has a drive error.';
	END_IF
	IF Cover2_error THEN 
		Covers_Error_Event.OnMessage := 'Cover 2 has a drive error.';
	END_IF
	IF Cover1_error  AND NOT GVL_Main.isRoboTel THEN 
		Covers_Error_Event.OnMessage := 'Cover 1 has a drive error.';
	END_IF
END_IF

Covers_Error_event(	Trigger := Error, 
					Level := ADSLOG_MSGTYPE_ERROR);

Covers_Warning_event(	Trigger := Warning, 
						Level := ADSLOG_MSGTYPE_WARN);

// raise an error, if both opened and closed signals are activated
// handle RoboTel differently
Cover1_Event(	Trigger := cover1_opened AND cover1_closed AND NOT GVL_Main.isRoboTel,
				Level := ADSLOG_MSGTYPE_ERROR, 
				OnMessage := 'Cover1: limit switch error');

Cover2_Event(Trigger := cover2_opened AND cover2_closed,
				Level := ADSLOG_MSGTYPE_ERROR, 
				OnMessage := 'Cover2: limit switch error');

Cover3_Event(Trigger := cover3_opened AND cover3_closed,
				Level := ADSLOG_MSGTYPE_ERROR, 
				OnMessage := 'Cover3: limit switch error');

//trigger an event, if we encounter a timeout
// handle RoboTel differently

Cover1_Timeout_Event(Trigger := FALSE,
				Level := ADSLOG_MSGTYPE_ERROR, 
				OnMessage := 'Cover1: Timeout');

Cover2_Timeout_Event(Trigger := FALSE,
				Level := ADSLOG_MSGTYPE_ERROR, 
				OnMessage := 'Cover2: Timeout');

Cover3_Timeout_Event(Trigger := FALSE,
				Level := ADSLOG_MSGTYPE_ERROR, 
				OnMessage := 'Cover3: Timeout');
// Log if we are opened
Covers_opened_event(Trigger := isopen,
					Level := ADSLOG_MSGTYPE_WARN,
					OnMessage := 'All covers are open');
//log if we are closed
Covers_closed_event(Trigger := isclosed,
					Level := ADSLOG_MSGTYPE_HINT,
					OnMessage := 'All covers are closed');

END_PROGRAM

// ---- POUs/FocusControl.TcPOU
PROGRAM FocusControl
VAR_INPUT
	// enable the axis
	enable: BOOL;
	// Move M2 closer to M1
	inward: 	BOOL;
	// Move M2 away from M1
	outward: 	BOOL;	
	// reset the axis(-error)
	reset: 		BOOL;
	// move the axis to new position
	MoveAxis:	BOOL;
	// calibrate the focus axis
	HomeAxis:	BOOL;
	// focus position in millimeters
	position: 		LREAL;
END_VAR

VAR_OUTPUT
	// true if absolute calibration
	Calibrated:	BOOL;
	// true if error
	Error: 		BOOL;
	// ID of NC axis error
	ErrorID:	UDINT;
	// ready signal = drive ready + standstill
	Ready:	BOOL;
END_VAR

VAR
	FocusDelay:			TON;
	BrakeDelay:			TON;
	FocusAxis:			FB_Axis2;
	actual_position:	LREAL;
	// manual override to unlock the focus
	FocusUnlock:		BOOL;
	FocusUnlocked:		BOOL;
	MQTTTimer : 		TON := (PT:=T#5S);
	//getlastposition:	BOOL := TRUE;
	FocusAxisEvent:		FB_EventLog;
	CalibrationEvent:	FB_EventLog;
	HomingMode: 		MC_HOMINGMODE := 		MC_DefaultHoming;
	SetPosition:		MC_SetPosition;
END_VAR

VAR CONSTANT
	// reference position for homing
	homing_position:		LREAL := 92.8936; // 106.5936 - 13.7000
	tolerance:				LREAL := 0.005;
END_VAR
VAR PERSISTENT
	last_position:		LREAL := -1.0;
END_VAR

(*
Focus Control Unit
spindle gear: 5mm
brake: 86 61103H00 Var. 0005 Index C; 24VDC geglattet 0,25 A P1672/R7
motor: Faulhaber ; Schönaich ; 3557K024CR; 454  431 ; Made in germany ==> 5300 rpm
gear: Faulhaber ; MINIMOTOR SA ; swiss made ; 38/1S  43:1 ; 033896  503
Focus is locked by default
70,8W; 0,100A no load current; 2,0 Terminal resistance; 1,950A max Current 
*)
position := LIMIT(5.0, position, 95.0);

GVL_Telescope.focus_unlock := FocusUnlock OR enable;

// wait until the focus is unlocked for n milliseconds
FocusDelay(IN := GVL_Telescope.focus_unlock, PT := T#500MS, Q => FocusUnlocked);
// wait for brake until we are at rest
BrakeDelay(IN := NOT FocusAxis.Busy AND FocusAxis.StandStill, PT := T#4000MS);

// if we are on automatic mode then position the focus
IF Pendantcontrol.telescope_mode = E_TelescopeMode.automatic AND NOT FocusUnlock THEN
	IF FocusAxis.Calibrated THEN
		IF ABS(position - actual_position) > tolerance THEN
			IF FocusAxis.Ready THEN
				MoveAxis := TRUE;
			ELSE
				Enable := TRUE;
			END_IF
		END_IF
		// disable the drive and lock the brake, if we stand for more than n seconds
		IF BrakeDelay.Q THEN
			Enable := FALSE;
		END_IF
		// store actual position, if we are calibrated and locked
		IF NOT GVL_Telescope.focus_unlock THEN
			last_position := actual_position;
		END_IF
	ELSE // not calibrated
		IF FocusAxis.Ready THEN
			HomeAxis := TRUE;
		END_IF
	END_IF
END_IF

IF HomeAxis THEN
	IF last_position > 0.0 THEN
		HomingMode := MC_ForceCalibration; // MC_Direct
		position := last_position;
		SetPosition.Execute := TRUE;
	ELSE
		HomingMode := MC_DefaultHoming;
		position := homing_position;
		SetPosition.Execute := FALSE;
	END_IF
ELSE
	SetPosition.Execute := FALSE;	
END_IF

// deactivate limit switches on homing
MC_SetAcceptBlockedDriveSignal(
	Axis := GVL_Telescope.FocusAxisRef, 
	Enable := HomeAxis);
SetPosition(
	Axis := GVL_Telescope.FocusAxisRef, 
	Position := last_position);
	
	
FocusAxis(	
	Enable := 			FocusUnlocked,
	Reset := 			reset,
	MoveAxis := 		MoveAxis AND FocusUnlocked,
	HomeAxis :=			HomeAxis AND FocusUnlocked,
	HomingMode :=		HomingMode,
	Position := 		position,
	Velocity :=			0.02,
	Enable_Positive := 	NOT GVL_Telescope.focus_limit_far OR HomeAxis,
	Enable_Negative := 	NOT GVL_Telescope.focus_limit_near,
	Jog_Forward :=		outward AND FocusUnlocked,
	Jog_Backwards := 	inward AND FocusUnlocked,
	bCalibrationCam :=  GVL_Telescope.focus_limit_far,
	ActualPosition => 	actual_position,
	Error =>			error,
	ErrorID =>			ErrorID,
	AxisRef :=			GVL_Telescope.FocusAxisRef);	

IF FocusAxis.MoveDone THEN
	MoveAxis := FALSE;
END_IF

IF FocusAxis.HomeDone THEN
	HomeAxis := FALSE;
	Enable := FALSE;
	last_position := position;
END_IF
	
IF FocusAxis.ResetDone THEN
	reset := FALSE;
END_IF

IF FocusAxis.Calibrated OR Error THEN
	HomeAxis := FALSE;
END_IF

IF Error THEN
	last_position := -1.0;
	//FocusAxis.Calibrated := FALSE;
	Calibrated := FALSE;
END_IF

Calibrated := FocusAxis.Calibrated;

Ready := FocusAxis.Ready AND FocusAxis.StandStill OR NOT GVL_Telescope.focus_unlock;

MQTTTimer(IN:=TRUE);
IF MQTTTimer.Q THEN // publish new payload every second
	MQTTTimer(IN:=FALSE);
	MAIN.MQTTClient.Publish('telescope', 'dome', 'FocusPosition', LREAL_TO_FMTSTR(actual_position, 5, TRUE));
	MAIN.MQTTClient.Publish('telescope', 'dome', 'FocusCalibrated', BOOL_TO_STRING(Calibrated));	
	MAIN.MQTTClient.Publish('telescope', 'dome', 'FocusReady', BOOL_TO_STRING(Ready));	
END_IF

FocusAxisEvent(	
	Trigger := 		FocusAxis.Error, 
	Level := 		ADSLOG_MSGTYPE_ERROR,
	FormatString :=	'Focus Axis Error: %s',
	OnMessage := 	NCError_TO_STRING(ErrorID),
	OffMEssage := 	'OK',
	OffLevel := 	ADSLOG_MSGTYPE_HINT);

CalibrationEvent(
	Trigger :=	Calibrated,
	Level :=	ADSLOG_MSGTYPE_HINT,
	OnMessage := 'Focus is calibrated.'
	);

END_PROGRAM

// ---- POUs/PendantControl.TcPOU
PROGRAM PendantControl
VAR_IN_OUT
	CoverControl	: FB_CoverControl;
	HydraulicsControl : FB_HydraulicsControl;
	Focuscontrol : FB_Focuscontrol;
	DerotatorControl	: FB_DerotatorControl;
	ElevationControl	: FB_ElevationControl;
	AzimuthControl : FB_AzimuthControl;
END_VAR
VAR_INPUT
	comm: I_Comm;
END_VAR
VAR
	// program selection of the pendant control
	Selection:	UINT;
	// error on the pendant control
	Error:		BOOL;
	// manual switch
	manual:		BOOL;
	//enable button
	enable:		BOOL;
	//reset button
	reset:		BOOL;
	// up button
	up:			BOOL;
	// down button
	down:		BOOL;
	// left button
	left:		BOOL;
	// right button
	right:		BOOL;
	lamp_left:		BOOL;
	lamp_right:		BOOL;
	lamp_up:		BOOL;
	lamp_down:		BOOL;
	lamp_error:		BOOL;
	horn:			BOOL;
	FocusEnable: 		FB_ButtonEnable;
	DerotatorEnable:	FB_ButtonEnable;
	ElevationEnable: 	FB_ButtonEnable;
	AzimuthEnable: 		FB_ButtonEnable;
	TelescopeControlEnable: 	FB_ButtonEnable;
	HydraulicsEnable: 	FB_ButtonEnable;
	TrackingEnable:			FB_ButtonEnable;
	ResetDelay:	TON;
	TwinCATRestart: TC_Restart;
	up_trigger:	R_TRIG;
	down_trigger:	R_TRIG;	
	// manual or automatic operation of the telescope
	telescope_mode : E_TelescopeMode;	
END_VAR

(* 
This program is responsible for the manual control of the telescope.
all movable parts can be controlled from here. This is mainly for testing and
maintenance.
WARNING! Some of the safety routines are disabled, when operating the telescope manually.
*)
// calculate the value of the selector
Selection := 1*BOOL_TO_UINT(GVL_pendant_control.BCD1) + 
			 2*BOOL_TO_UINT(GVL_pendant_control.BCD2) + 
			 4*BOOL_TO_UINT(GVL_pendant_control.BCD4) +
			 8*BOOL_TO_UINT(GVL_pendant_control.BCD8);

// detect disconnection of the manual controls (should also trigger emergency stop).			 
Error := (Selection = 0);

// disable all the lamps
lamp_left := FALSE;
lamp_right := FALSE;
lamp_up := FALSE;
lamp_down := FALSE;
horn := FALSE;

// clooect the state of all buttons
manual := GVL_pendant_control.key_switch;
enable := GVL_pendant_control.start_switch;
reset := GVL_pendant_control.reset_switch;
up := GVL_pendant_control.direction_up;
down := GVL_pendant_control.direction_down;
left := GVL_pendant_control.direction_left;
right := GVL_pendant_control.direction_right;

up_trigger(CLK := up);
down_trigger(CLK := down);
//R_Enable(CLK := enable);
// the error lamp is the same as the error lamp of the main panel
lamp_error := GVL_Main.lamp_error;


// determine the operation of the telescope based on the switch set
IF manual THEN
	telescope_mode := E_TelescopeMode.manual;
ELSE
	telescope_mode := E_TelescopeMode.automatic;
END_IF

// enable only the selected item and connect lamps and buttons accordingly
CASE Selection OF
	1:	// reserved for Cover1 control
		lamp_up := CoverControl.cover1_open;
		lamp_down := CoverControl.cover1_closed;
		IF manual THEN
			//CoverEnable(SET := enable, Q := CoverControl.enable);
			//CoverControl.active_cover := 1;
			//CoverControl.reset := reset;
			CoverControl.open_cover1 := up AND CoverControl.cover1_open;
			CoverControl.close_cover1 := down AND CoverControl.cover1_closed;
			lamp_error := CoverControl.Cover1_Error;	
		ELSE
			IF down THEN 
				CoverControl.close := TRUE;
			END_IF
			IF up THEN
				CoverControl.open := TRUE;
			END_IF		
		END_IF

	2: // Cover2 control
		lamp_up := CoverControl.cover2_open;
		lamp_down := CoverControl.cover2_closed;
		IF manual THEN
			//CoverEnable(SET := enable, Q := CoverControl.enable);
			//CoverControl.active_cover := 2;
			CoverControl.open_cover2 := up AND CoverControl.cover2_open;
			CoverControl.close_cover2 := down AND CoverControl.cover2_closed;
			lamp_error := CoverControl.Cover2_Error;
		ELSE
			IF down THEN 
				CoverControl.close := TRUE;
			END_IF
			IF up THEN
				CoverControl.open := TRUE;
			END_IF		
		END_IF
 	
	3:  // Cover3 control
		lamp_up := CoverControl.cover3_open;
		lamp_down := CoverControl.cover3_closed;
		IF manual THEN
			//CoverEnable(SET := enable, Q := CoverControl.enable);
			//CoverControl.active_cover := 3;
			CoverControl.open_cover3 := up AND CoverControl.cover3_open;
			CoverControl.close_cover3 := down AND CoverControl.cover3_closed;
			//CoverControl.reset := reset;
			lamp_error := CoverControl.Cover3_Error;
		ELSE
			IF down THEN 
				CoverControl.close := TRUE;
			END_IF
			IF up THEN
				CoverControl.open := TRUE;
			END_IF		
		END_IF
		
	4:	// Nasmyth / mirror M3 control
		
	5:	// Focus Control
		lamp_up := FocusControl.Ready AND NOT FocusControl.limitFar;
		lamp_down := FocusControl.Ready AND NOT FocusControl.limitNear;
		IF manual THEN
			FocusEnable(SET := enable, Q := FocusControl.enable);
			FocusControl.outward := up;
			FocusControl.inward := down;
			Focuscontrol.reset := reset;
			lamp_error := FocusControl.error;
		END_IF
							
	6:	// Derotator control
		lamp_left := DerotatorControl.Ready AND NOT DerotatorControl.digital_inputs.1;
		lamp_right :=DerotatorControl.Ready AND NOT DerotatorControl.digital_inputs.0;
		IF manual THEN
			DerotatorEnable(SET := enable, Q := DerotatorControl.enable);
			DerotatorControl.left := left AND NOT DerotatorControl.digital_inputs.1;
			DerotatorControl.right := right AND NOT DerotatorControl.digital_inputs.0;
			DerotatorControl.reset := reset;
			lamp_error := DerotatorControl.Error;
		END_IF
							
	7:	// Elevation Control
		
		ElevationControl.up := up AND ElevationControl.digital_inputs.0;
		ElevationControl.down := down AND ElevationControl.digital_inputs.1;
		IF manual THEN
			ElevationEnable(
				SET := enable, 
				Q := ElevationControl.enable);	
		END_IF
		ElevationControl.reset := reset;
		lamp_up := ElevationControl.digital_inputs.0;
		lamp_down := ElevationControl.digital_inputs.1;
		lamp_error := ElevationControl.error;
		
	8:	// Azimuth Control
		lamp_left := AzimuthControl.digital_inputs.0; // NOT GVL_Telescope.azimut_limit_switch;
		lamp_right := AzimuthControl.digital_inputs.1; // NOT GVL_Telescope.azimut_limit_switch;
		AzimuthControl.left := left AND AzimuthControl.digital_inputs.0;
		AzimuthControl.right := right AND AzimuthControl.digital_inputs.1;
		AzimuthControl.reset := reset;
		IF manual THEN
			AzimuthEnable(
				SET := enable, 
				Q := AzimuthControl.enable);
			lamp_error := AzimuthControl.error;
		END_IF
		
	9: 	// Dome control
		
	10:	// FilterWheel control
		
	11: lamp_up := ElevationControl.elevation_torque > 0.0;
		lamp_down := ElevationControl.elevation_torque < 0.0;
		
	12:	// manual Telescope Control
		IF manual THEN
			lamp_up := TelescopeControl.power;
			lamp_down := TelescopeControl.power;
			lamp_left := TelescopeControl.power;
			lamp_right := TelescopeControl.power;
	
			TelescopeControl.gohome := down;
			TelescopeControl.park := up;
			TelescopeControl.goto := right;
			TrackingEnable(SET := enable, 
							RESET := reset, 
							Q := TelescopeControl.track);
			TelescopeControl.reset := reset;
			Telescopecontrol.stop := left;	
			lamp_error := Telescopecontrol.error;
		END_IF
		
	13: // Telescope Control
		TelescopeControlEnable(
			SET := enable, 
			Q := TelescopeControl.power);
		TelescopeControl.reset := reset;
		IF manual THEN
			lamp_up := ElevationControl.digital_inputs.0;
			lamp_down := ElevationControl.digital_inputs.1;
			lamp_left := AzimuthControl.digital_inputs.0;
			lamp_right := AzimuthControl.digital_inputs.1;
			ElevationControl.up := up AND ElevationControl.digital_inputs.0;
			ElevationControl.down := down AND ElevationControl.digital_inputs.1;
			AzimuthControl.left := left AND AzimuthControl.digital_inputs.0;
			AzimuthControl.right := right AND AzimuthControl.digital_inputs.1;
			TelescopeControl.rightascension := TelescopeControl.rightascension_calc;
			TelescopeControl.declination := TelescopeControl.declination_calc;
		ELSE
			lamp_up := ElevationControl.enable;
			lamp_down := ElevationControl.enable;
			lamp_left := AzimuthControl.enable;
			lamp_right := AzimuthControl.enable;
			IF up THEN 
				Telescopecontrol.elevation_offset := Telescopecontrol.elevation_offset + 10.0/3600.0; 
			ELSIF down THEN 
				Telescopecontrol.elevation_offset := Telescopecontrol.elevation_offset - 10.0/3600.0; 
			END_IF;
			IF left THEN 
				Telescopecontrol.azimuth_offset := Telescopecontrol.azimuth_offset - 10.0/3600.0; 
			ELSIF right THEN 
				Telescopecontrol.azimuth_offset := Telescopecontrol.azimuth_offset + 10.0/3600.0; 
			END_IF;
		END_IF
		ResetDelay(IN := reset, PT := T#3S);
		// wait for suction pump to stop
		TwinCATRestart(NETID := '', RESTART := ResetDelay.Q AND NOT HydraulicsControl.suction_running, TMOUT := T#60S);
	
	14: horn := manual;
		lamp_up := manual;
		lamp_down := manual;
		lamp_left := manual;
		lamp_right := manual;
	
	15:	// Hydraulics control
		lamp_up := HydraulicsControl.oil_pressure_OK AND Hydraulicscontrol.brake_closed;
		lamp_down := HydraulicsControl.oil_pressure_OK AND Hydraulicscontrol.brake_open;
		lamp_left := HydraulicsControl.pump_running;
		lamp_right := HydraulicsControl.suction_running;
		IF manual THEN
			HydraulicsEnable(
				SET := enable, 
				Q := Hydraulicscontrol.enable);
			Hydraulicscontrol.reset := reset;
			
			IF up THEN
				Hydraulicscontrol.open_brake();
			END_IF
			IF down THEN
				Hydraulicscontrol.close_brake();
			END_IF
			Hydraulicscontrol.suction_manual := right;
			Hydraulicscontrol.pump_manual_stop := left;
			lamp_error := HydraulicsControl.error;
		END_IF
END_CASE

// set all the lamps
GVL_pendant_control.lamp_left := lamp_left;
GVL_pendant_control.lamp_right := lamp_right;
GVL_pendant_control.lamp_up := lamp_up;
GVL_pendant_control.lamp_down := lamp_down;
GVL_pendant_control.lamp_error := lamp_error;

END_PROGRAM

// ---- POUs/DerotatorControl.TcPOU
PROGRAM DerotatorControl
VAR_INPUT
	// enable the derotator
	enable:		BOOL;
	// reset an error
	reset:		BOOL;
	// decrease derotator angle
	left:		BOOL;
	// increase derotator angle
	right:		BOOL;
	// set the absolute position
	position:	LREAL;
	// derotator velocity
	Velocity:	LREAL := 10.0;
	// move to given position
	MoveAxis: 	BOOL;
	// calibrate the axis
	HomeAxis:	BOOL;
	// tracking flag
	Tracking:	BOOL;
	// stop the Axis
	StopAxis:	BOOL;
	// diagnostic error code reset
	bSoEReset: 			BOOL;
END_VAR
VAR_OUTPUT
	// error flag
	Error:				BOOL;
	// nc error id
	ErrorID:			UDINT;
	// actual position of the derotator
	actual_position:	LREAL;
	// calibrated flag
	Calibrated:			BOOL;
	// axis ready flag
	Ready:				BOOL;
	// position to move the axis to
	slewtime: 			LREAL;
END_VAR
VAR
	// trigger for the torque error
	TorqueError:		TON := (PT := T#3S);
	// axis function block
	DerotatorAxis:		FB_Axis2;
	
	DerotatorEvent:		FB_EventLog;
	// torque warning event
	TorqueWarning:		FB_EventLog;
	// torque calibration event
	CalibrationEvent:	FB_EventLog;
	// diagnostic low-level event
	DerotatorDiagnosticEvent: FB_EventLog;
	// percentage of the derotator torque
	derotator_torque:	REAL;
	// read slewtime
	ReadParameter:		MC_ReadParameter;
	fbSoEReset: 		FB_SoEReset;
	DiagnosticError:	BOOL;
END_VAR
VAR CONSTANT
	// current position of the calibration cam. Apply an offset here if necessary
	calibration_position:	LREAL := 438.4623; // calibration in positive direction (was 460.0)
END_VAR

(*
Selection 6
Homing in Endlage:

https://infosys.beckhoff.com/index.php?content=../content/1031/ax5000_usermanual/html/ax5000_homing_hardware_end_position.htm&id=12221
NC-Interface:
PlcToNc-Achsinterface, Bit 8 namens AcceptBlockedDriveSignal im nDeCtrlDWord

SPS-Interface:
TcNc-Lib, siehe SPS-Funktion AxisSetAcceptBlockedDriveSignal in der TwinCAT  PLC Library: NC.
*)

position := LIMIT(-70, position, 380);

IF enable AND NOT DerotatorAxis.Calibrated THEN
	HomeAxis := TRUE;
END_IF

IF DerotatorAxis.Calibrated THEN
	HomeAxis := FALSE;
	Calibrated := DerotatorAxis.Calibrated;
END_IF
	
IF HomeAxis THEN
	position := calibration_position;
END_IF

DeRotatorAxis(
	enable := 			enable,
	Reset := 			Reset,
	MoveAxis :=			MoveAxis,
	HomeAxis :=			HomeAxis,
	StopAxis :=			StopAxis,
	HomingMode :=		MC_ForceCalibration,
	Position := 		position, 
	Velocity :=			Velocity,
	Enable_Positive := 	NOT GVL_Telescope.Derotator_inputs.0,
	Enable_Negative := 	NOT GVL_Telescope.Derotator_inputs.1,
	Jog_Forward := 		right,
	Jog_Backwards := 	left,
	bCalibrationCam :=	GVL_Telescope.Derotator_inputs.0,
	isModuloAxis :=		FALSE,
	Tracking :=			Tracking,
	ActualPosition => 	actual_position,
	Error => 			Error,
	ErrorID => 			ErrorID,
	AxisRef :=			GVL_Telescope.DerotatorAxisRef);
	
IF DeRotatorAxis.MoveDone OR Reset OR Error THEN
	MoveAxis := FALSE;
END_IF

IF DeRotatorAxis.HomeDone OR Reset OR Error THEN
	HomeAxis := FALSE;
END_IF
	
IF DeRotatorAxis.ResetDone THEN
	reset := FALSE;
END_IF

IF DeRotatorAxis.StopDone THEN
	StopAxis := FALSE;
END_IF

DiagnosticError := FALSE;
IF GVL_Telescope.Derotator_diagnostic < 16#D012 AND GVL_Telescope.Derotator_diagnostic > 16#D014 THEN
	DiagnosticError := TRUE;
	ErrorID := GVL_Telescope.Derotator_diagnostic;
	bSoeReset := reset;
END_IF

Ready := DeRotatorAxis.Ready;

ReadParameter(	Axis := GVL_Telescope.DerotatorAxisRef, 
				Enable := DeRotatorAxis.InMotion, 
				ParameterNumber := MC_AxisParameter.AxisRemainingTimeToGo, 
				ReadMode := E_ReadMode.READMODE_CYCLIC);
				
IF ReadParameter.Valid THEN
	slewtime := ReadParameter.Value;
END_IF

IF bSoEReset THEN
	fbSoEReset(
		Axis := GVL_Telescope.DerotatorAxisRef,
		Execute := TRUE,
		Timeout := DEFAULT_ADS_TIMEOUT);
 	IF NOT fbSoEReset.Busy THEN
		fbSoEReset(Axis := GVL_Telescope.DerotatorAxisRef, Execute := FALSE);
		bSoEReset := FALSE;
		Reset := TRUE;
	END_IF
END_IF

derotator_torque := GVL_Telescope.Derotator_torque / 10.0;
// nominal torque is 3%, max is 25%
TorqueError(IN := ABS(derotator_torque) > 20.0);

DerotatorEvent(	
	Trigger := 		Error, 
	Level := 		ADSLOG_MSGTYPE_ERROR,
	FormatString :=	'Derotator Axis Error: %s',
	OnMessage := 	NCError_TO_STRING(ErrorID),
	OffMEssage := 	'OK',
	OffLevel := 	ADSLOG_MSGTYPE_HINT);
	
DerotatorDiagnosticEvent(	
	Trigger := 		DiagnosticError, 
	Level := 		ADSLOG_MSGTYPE_ERROR,
	FormatString :=	'Derotator Axis Diagnostic Error: %s',
	OnMessage := 	NCError_TO_STRING(GVL_Telescope.Derotator_diagnostic));
	
TorqueWarning(	
	Trigger := 		TorqueError.Q, 
	Level := 		ADSLOG_MSGTYPE_WARN,
	FormatString :=	'%s',
	OnMessage := 	'Derotator torque is high.');

CalibrationEvent(	
	Trigger := 		Calibrated, 
	Level := 		ADSLOG_MSGTYPE_HINT,
	OnMessage := 	'Derotator is calibrated.');

END_PROGRAM

// ---- POUs/ElevationControl.TcPOU
PROGRAM ElevationControl
VAR_INPUT
	// enable the axis
	enable: 	BOOL;
	// reset an error
	reset:		BOOL;
	// increase the eleveation
	up:			BOOL;
	// decrease the elevation
	down:		BOOL;
	// set position of the axis in degrees
	position:	LREAL;
	// set the Velocity of the axis
	velocity:	LREAL;
	// move axis command
	MoveAxis:	BOOL;
	// calibrate the axis
	HomeAxis:	BOOL;
	// enable tracking
	Tracking:	BOOL;
	// stop the Axis
	StopAxis:	BOOL;
	// reset diagnostic errors
	bSoEReset:	 	BOOL;
	comm : I_Comm;
END_VAR
VAR_IN_OUT	
	CoverControl	: FB_CoverControl;
	HydraulicsControl : FB_HydraulicsControl;
END_VAR
VAR_OUTPUT
	// axis is ready to operate
	Ready:			BOOL;
	// drive error condition
	error: 			BOOL;
	// warning condition
	warning:		BOOL;
	// actual position of the elevation axis
	actual_position: 	LREAL;
	// error ID of the elevation axis
	ErrorID: 		UDINT;
	// axis is calibrated
	Calibrated:		BOOL;
	// time to reach target position
	slewtime:		LREAL;
END_VAR
VAR
	ElevationAxis:			FB_Axis2;
	ElevationCalibration: 	MC_SetPosition;
	fbSoEReset: 			FB_SoEReset;
	// delay until commutator angle is measured
	readydelay:				TON;
	// disable trigger for hydraulics
	enable_trigger:			F_TRIG;
	// store last position
	getlastposition:		BOOL := TRUE;
	ElevationAxisEvent: 	FB_Eventlog;
	ElevationDiagnosticEvent: 	FB_Eventlog;
	ElevationBrakeEvent: 	FB_Eventlog;
	HighElevationEvent: 	FB_Eventlog;
	LowElevationEvent:		FB_Eventlog;
	TorqueWarning:			FB_EventLog;
	CalibrationEvent:		FB_Eventlog;
	// elevation torque in percent
	elevation_torque: 		REAL;
	// timer to trigger a warning if torque is high
	torque_timer:			TON;
	ReadParameter:			MC_ReadParameter;
	DiagnosticError:		BOOL;
END_VAR
VAR CONSTANT
	// current position of the calibration cam. Apply an offset here if necessary
	calibration_position:	LREAL := 44.144; //44.139; //44.061; //43.806122; //42.1281; //43.000
END_VAR
VAR PERSISTENT
	last_position:	LREAL := -1.0;
END_VAR

// limit the position input to a sane value
position := LIMIT(0.0, position, 90.0);

//if we enable the axis, we have to open the brake first
IF Enable THEN
	IF NOT Calibrated THEN
		CoverControl.open := TRUE;
		IF CoverControl.isopen THEN
			HydraulicsControl.open_brake();
		END_IF
	ELSE
		HydraulicsControl.open_brake();
	END_IF
	
END_IF

enable_trigger(CLK := enable);
// close the brake on the falling edge of the enable signal
IF enable_trigger.Q THEN
	HydraulicsControl.close_brake();
END_IF

IF ElevationAxis.Calibrated OR Error THEN
	HomeAxis := FALSE;
END_IF

Calibrated := ElevationAxis.Calibrated;

IF HomeAxis THEN
	position := calibration_position;
	MoveAxis := FALSE;
	Tracking := FALSE;
END_IF

IF MoveAxis THEN
	Tracking := FALSE;
END_IF

// if NOT Enabled and ActVelo>1 then issue a warning
warning := NOT enable AND GVL_Telescope.ElevationAxisRef.NcToPlc.ActVelo>2.0;

// deactivate limit switches on homing
MC_SetAcceptBlockedDriveSignal(
	Axis := GVL_Telescope.ElevationAxisRef, 
	Enable := HomeAxis);
	
ElevationAxis(
	Enable := 			enable AND HydraulicsControl.brake_open,
	Reset := 			reset,
	MoveAxis :=			MoveAxis,
	HomeAxis :=			HomeAxis,
	StopAxis :=			StopAxis,
	Tracking :=			Tracking,
	Position := 		position, 
	Velocity :=			Velocity,
	Enable_Positive :=  GVL_Telescope.Elevation_inputs.0 OR HomeAxis,
	Enable_Negative := 	GVL_Telescope.Elevation_inputs.1,
	Jog_Forward :=		up,
	Jog_Backwards := 	down,
	bCalibrationCam :=	NOT GVL_Telescope.Elevation_inputs.0,
	ActualPosition => 	actual_position,
	Error => 			error,
	ErrorID => 			ErrorID,
	AxisRef :=			GVL_Telescope.ElevationAxisRef);

IF ElevationAxis.MoveDone THEN
	MoveAxis := FALSE;
END_IF

IF ElevationAxis.HomeDone THEN
	HomeAxis := FALSE;
END_IF
	
IF ElevationAxis.ResetDone THEN
	reset := FALSE;
END_IF

IF ElevationAxis.StopDone THEN
	StopAxis := FALSE;
END_IF

DiagnosticError := FALSE;
IF GVL_Telescope.Elevation_diagnostic < 16#D012 AND GVL_Telescope.Elevation_diagnostic > 16#D014 THEN
	DiagnosticError :=TRUE;
	ErrorID := GVL_Telescope.Elevation_diagnostic;
END_IF

ElevationCalibration(Axis := GVL_Telescope.ElevationAxisRef,
	Execute := getlastposition AND last_position>=0.0 AND NOT Calibrated,
	Position := last_position);

IF ElevationCalibration.Done THEN
	getlastposition := FALSE;
END_IF

IF Calibrated THEN
	last_position := actual_position;
END_IF

IF bSoEReset THEN
	last_position := -1.0;
	fbSoEReset(
		Axis := GVL_Telescope.ElevationAxisRef,
		Execute := TRUE,
		Timeout := DEFAULT_ADS_TIMEOUT);
 	IF NOT fbSoEReset.Busy THEN
		fbSoEReset(Axis := GVL_Telescope.ElevationAxisRef, Execute := FALSE);
		bSoEReset := FALSE;
		Reset := TRUE;
	END_IF
END_IF 

readydelay(IN :=  HydraulicsControl.brake_open, PT := T#6000MS, Q=> ready);

ReadParameter(	Axis := GVL_Telescope.ElevationAxisRef, 
				Enable := ElevationAxis.InMotion, 
				ParameterNumber := MC_AxisParameter.AxisRemainingTimeToGo, 
				ReadMode := E_ReadMode.READMODE_CYCLIC);
				
IF ReadParameter.Valid THEN
	slewtime := ReadParameter.Value;
END_IF

elevation_torque := GVL_Telescope.Elevation_torque / 10.0;
torque_timer(IN := ABS(elevation_torque) > 50.0, PT := T#1000MS);
		
ElevationAxisEvent(	Trigger := Error, 
				Level := ADSLOG_MSGTYPE_ERROR,
				FormatString := 'Elevation Axis Error: %s',
				OnMessage := NCError_TO_STRING(ErrorID), 
				Comm := comm);

ElevationDiagnosticEvent(	
	Trigger := 		DiagnosticError, 
	Level := 		ADSLOG_MSGTYPE_ERROR,
	FormatString :=	'Elevation Axis Diagnostic Error: %s',
	OnMessage := 	NCError_TO_STRING(GVL_Telescope.Elevation_diagnostic), 
	Comm := comm);

				
HighElevationEvent(	Trigger := Calibrated AND actual_position > 85.0, 
				Level := ADSLOG_MSGTYPE_WARN,
				FormatString := 'High Elevation: %s',
				OnMessage := LREAL_TO_FMTSTR(actual_position, 2, TRUE), 
				Comm := comm);

LowElevationEvent(	Trigger := Calibrated AND actual_position < 5.0, 
				Level := ADSLOG_MSGTYPE_WARN,
				FormatString := 'Low Elevation: %s',
				OnMessage := LREAL_TO_FMTSTR(actual_position, 2, TRUE), 
				Comm := comm);
				
ElevationBrakeEvent( Trigger := NOT enable AND HydraulicsControl.brake_open, 
				Level := ADSLOG_MSGTYPE_WARN,
				FormatString := '%s',
				OnMessage := 'Brake was opened without elevation axis enabled!', 
				Comm := comm); 

TorqueWarning(	
	Trigger := torque_timer.Q, 
	Level := 		ADSLOG_MSGTYPE_WARN,
	FormatString :=	'%s',
	OnMessage := 	'Elevation torque is high.', 
				Comm := comm);
	
CalibrationEvent(
	Trigger :=	Calibrated,
	Level :=	ADSLOG_MSGTYPE_HINT,
	OnMessage := 'Elevation is calibrated.', 
				Comm := comm);

END_PROGRAM

// ---- POUs/TelescopeControl.TcPOU
PROGRAM TelescopeControl
VAR_INPUT
(*
TCS interface section
see https://gitlab.aip.de/bmk10k/telescope_firmware/snippets/5
*)
	
	// boolean, true: Power on, false: power off
	power: 		BOOL;
	// boolean, true: go to home position, unset track/goto if active
	gohome: 	BOOL;
	// boolean, true: go into park position, ready to stow telescope, unset track/goto
	park: 		BOOL;
	// boolean, TRUE: MOVE telescope TO last ra/de AND start tracking. Set 'goto' TO FALSE, IF TRUE. FALSE: Stop tracking as soon as possible
	track: 		BOOL;
	// boolean, TRUE: MOVE telescope TO tau/de AND stop there. Set track TO FALSE, IF TRUE. FALSE: no effect.)
	goto:		BOOL;	
	// move the telescope to a given az-alt position
	slew:		BOOL;
	// boolean, TRUE: Stop motion OF telescope immediately, set goto AND track TO FALSE. FALSE: Allow motion OF telescope again via track/goto).
	stop:		BOOL;	
	// initiates reset on all axis
	reset:		BOOL;
	// automatic tracking after goto
	autotrack:	BOOL := TRUE;
	// apparent right ascension, degrees, double
	rightascension:		LREAL := (4.0 + 35.0/60.0 + 54.09/3600.0) *15.0;	
	// apparent declination, degrees, double
	declination: 		LREAL := 16.0 + 30.0/60.0 + 25.4/3600.0;
	// desired elevation of the telescope pointing 
	elevation:	LREAL := 45.0;
	// desired azimut of the telescope pointing 
	azimuth:	LREAL := 320.0;
	// absolute offset for elevation
	elevation_offset:	LREAL := 0.0;
	// absolute offset for azimuth
	azimuth_offset : 	LREAL := 0.0;
	// absolute offset for time
	time_offset: 		LREAL := 0.0;
	// offset for the de-rotator
	derotator_offset:	LREAL := 0.0;
END_VAR
VAR
	// actual command from the TCS
	TCS_command: 	E_TCSCommand;
	// current Julian Date calculated from system time
	jd:				LREAL;
	// image derotation
	derotation_calc:	LREAL;
	// local siderial time calculated from Julian date
	lst:			LREAL;
	// elevation calulated when ra and dec are set by TCS
	elevation_calc:	LREAL; 
	// azimuth calulated when ra and dec are set by TCS
	azimuth_calc:	LREAL;
	// right ascension calulated when azimuth and elevation are set by TCS
	rightascension_calc:	LREAL;
	// declination calulated when azimuth and elevation are set by TCS
	declination_calc:		LREAL;
	// hour angle
	Hourangle_calc: LREAL;
	// precise astronomical	time
	fbTime: FB_AstroClock;
	
	eq2hor:		FB_EQ2HOR;
	hor2eq:		FB_HOR2EQ;
	
	// triggers power-failure event
	powerfailure: 	BOOL;
	// triggers power warning
	poweronwarning:	TP;
	// power on timeout
	power_timeout:	TON;
	// command timeout
	command_timeout:	TON;
	// tracking delay
	tracking_delay:	TON;
	// telescope is parked
	isparked:		BOOL;
	TCSpowerEvent,
	TCSgohomeEvent,
	TCSparkEvent,
	TCSgotoEvent,
	TCStrackEvent,
	TCSstopEvent,
	AltitudeEvent,
	TCSreadyEvent,
	TCSCTOEvent: FB_Eventlog;
	MQTTTimer : TON := (PT:=T#5S);
	// rotational velocity of the derotator
	DerotatorVelocity: LREAL;
	// rotational velocity of the elevation
	ElevationVelocity: LREAL;
	// rotational velocity of the elevation
	AzimuthVelocity: LREAL;
	// sign of derotation
	derotatation_sign: LREAL := 1.0;
	StatusWord, LastStatus:	UDINT;
END_VAR
VAR_OUTPUT
	//		TRUE, IF telescope can be operated
	ready:		BOOL; 
	// indicates an error on one of the components
	error:		BOOL;	
	//error id of axis
	errorid:	UDINT;	
	//TRUE, IF telescope is in fast-MOVE phase (includes pole-swap)
	sliding:	BOOL;	
	//TRUE, IF telescope is on tracking position AND currently tracking.
	tracking:	BOOL;	
	//TRUE, IF telescope is AT rest.
	stopped:	BOOL;	
	// true position of the elevation
	elevation_current:	LREAL;
	// true position of the azimuth
	azimuth_current:	LREAL;
	// true position of the de-rotator
	derotator_current:	LREAL;
	//	(time in sec. to reach the goto/track position)
	slewtime:			LREAL; 
	// True: telescope is calibrated
	homed:				BOOL;
	// telescope does not accept further commands
	busy:				BOOL;
END_VAR
VAR CONSTANT
// STELLA1
	// telescope site longitude, source: Google 
	longitude: 		LREAL := -16.50926; //13.101867;
	// telescope site latitude, source: Google
	latitude: 		LREAL := 28.30120; //52.404940;
	// telescope site height above sea level: estimated
	altitude: 		LREAL := 2390.0;
	elevation_park: LREAL := 60.0;
	azimuth_park: 	LREAL := 359.999;
	derotator_park: LREAL := 229.85;

	elevation_home: LREAL := 55.0;
	azimuth_home: 	LREAL := 180.0;
END_VAR
VAR PERSISTENT
	// azimuth axis offset/misalignment north-south
	AN_E:	LREAL;
	// azimuth axis offset/misalignment east-west
	AE_E:	LREAL;
	// gravitational flexure correction at the horizon
	TF:		LREAL;
	// collimation error of the electromagnetic axis
	BNP:	LREAL;
	// azimuth axis offset/misalignment north-south
	AN_A:	LREAL;
	// azimuth axis offset/misalignment east-west,
	AE_A:	LREAL;
	// Non-perpendicularity between the mount azimuth and elevation axes
	NPAE:	LREAL;
END_VAR

TelescopeAuxiliary();

// get the system time
fbTime();
jd := DateTime2JD(fbTime.time_RTCEX2);
lst := CT2LST(longitude, jd);
// set reset state either by hardware (key pressed) or by software (set by e.g. tcs)
IF GVL_Main.reset_switch THEN
	reset := TRUE;
END_IF


IF ElevationControl.error THEN
	errorid := ElevationControl.ErrorID;
	ElevationControl.reset := reset;
ELSIF AzimuthElevationControl.error THEN
	errorid := AzimuthElevationControl.ErrorID;
	AzimuthElevationControl.Reset := reset;
ELSIF Focuscontrol.Error THEN
	errorid := Focuscontrol.ErrorID;
	FocusControl.reset := reset;
ELSIF DerotatorControl.Error THEN
	errorid := DerotatorControl.ErrorID;
	DerotatorControl.reset := reset;
END_IF

error := ElevationControl.error OR 
		 AzimuthElevationControl.error OR
		 Focuscontrol.Error OR
		 DerotatorControl.Error;

slewtime := MAX(MAX(ElevationControl.slewtime, AzimuthElevationControl.slewtime), DerotatorControl.slewtime);
			
IF error THEN
	gohome := 	FALSE;
	track := 	FALSE;
	goto := 	FALSE;
	slew := 	FALSE;
ELSE
	errorid := 0;
END_IF

IF ElevationControl.error THEN
	ElevationControl.enable := FALSE;
	AzimuthElevationControl.enable := FALSE;
	HydraulicsControl.close_brake();
END_IF

eq2hor(
	ra := rightascension,
	dec := declination,
	lon := longitude,
	lat := latitude,
	JD := jd + time_offset,
	alt => elevation_calc,
	az => azimuth_calc,
	ha => hourangle_calc);

// apply pointing model
elevation_calc := elevation_calc + PointingModelElevation(azimuth_calc, elevation_calc, elevation_offset, AN_E, AE_E, TF);
azimuth_calc := azimuth_calc + PointingModelAzimuth(azimuth_calc, elevation_calc, azimuth_offset, BNP, AN_A, AE_A, NPAE);
// calculate derotator position 
derotation_calc := F_DerotatorPosition2(azimuth_calc, elevation_calc, declination_calc, latitude, derotatation_sign)  + derotator_offset;
// calculate velocities
DerotatorVelocity := F_Derotatorvelocity(elevation_calc, azimuth_calc, latitude);
ElevationVelocity := F_Elevationvelocity(azimuth_calc, latitude);
AzimuthVelocity := F_Azimuthvelocity(elevation_calc, azimuth_calc, latitude);

IF (azimuth_calc > 310.0 AND AzimuthVelocity > 0.0) OR (azimuth_calc > 440.0) THEN
	azimuth_calc := azimuth_calc - 360.0;
ELSIF (azimuth_calc < 80.0 AND AzimuthVelocity < 0.0) OR (azimuth_calc < -50.0) THEN
	azimuth_calc := azimuth_calc + 360.0;
END_IF

IF (derotation_calc > 290.0 AND DerotatorVelocity > 0.0) OR (derotation_calc > 380.0) THEN
	derotation_calc := derotation_calc - 360.0;
ELSIF (derotation_calc < 20.0 AND DerotatorVelocity < 0.0) OR (derotation_calc < -70.0) THEN
	derotation_calc := derotation_calc + 360.0;
END_IF
// get current coordinates	
azimuth_current := AzimuthElevationControl.act_position;
elevation_current := ElevationControl.actual_position;
derotator_current := DerotatorControl.actual_position;

// calculate equatorial coordinates
hor2eq(alt := elevation_current - PointingModelElevation(azimuth_calc, elevation_calc, elevation_offset, AN_E, AE_E, TF), 
		az := azimuth_current - PointingModelAzimuth(azimuth_calc, elevation_calc, azimuth_offset, BNP, AN_A, AE_A, NPAE),
		jd := jd,
		lat := latitude,
		lon := longitude,
		altitude := altitude,
		ra => rightascension_calc,
		dec => declination_calc);		
	
poweronwarning(IN := power OR (NOT ElevationControl.enable AND HydraulicsControl.brake_open), PT := T#250MS);

power_timeout(IN := TCS_command = E_TCSCommand.no_command AND NOT isparked, PT := T#12H);
command_timeout();
IF power_timeout.Q AND NOT isparked THEN
	park := TRUE;
END_IF
		
// set TCS_command according to state variables ordered by precedence
IF power THEN
	TCS_command := E_TCSCommand.poweron;
ELSIF stop THEN
	TCS_command := E_TCSCommand.stop;
	goto := FALSE;
	track := FALSE;
	slew := FALSE;
	gohome := FALSE;
	park := FALSE;
ELSIF park THEN
	goto := FALSE;
	track := FALSE;
	slew := FALSE;
	IF ready AND stopped THEN
		TCS_command := E_TCSCommand.park;
	END_IF
ELSIF gohome THEN
	goto := FALSE;
	track := FALSE;
	slew := FALSE;
	IF ready AND NOT busy AND stopped THEN
		TCS_command := E_TCSCommand.gohome;
	END_IF
ELSIF goto THEN
	track := FALSE;
	slew := FALSE;
	IF ready AND NOT busy THEN
		TCS_command := E_TCSCommand.goto;
	END_IF
ELSIF slew THEN
	goto := FALSE;
	track := FALSE;
	IF ready AND NOT busy THEN
		TCS_command := E_TCSCommand.slew;
	END_IF
ELSIF track THEN
	goto := FALSE;
	slew := FALSE;
	IF ready AND NOT busy THEN
		TCS_command := E_TCSCommand.track;
	END_IF
ELSE
	TCS_command := E_TCSCommand.no_command;
	ElevationControl.MoveAxis := FALSE;
	AzimuthElevationControl.MoveAxis := FALSE;
	DerotatorControl.MoveAxis := FALSE;
	ElevationControl.Tracking := FALSE;
	AzimuthElevationControl.Tracking := FALSE;
	DerotatorControl.Tracking := FALSE;
END_IF

IF TCS_command = E_TCSCommand.poweron THEN
	poweron();
	command_timeout(IN := TCS_command = E_TCSCommand.poweron, PT := T#12H);
	TCSCTOEvent.OnMessage := 'POWER';
ELSIF TCS_command = E_TCSCommand.stop THEN
	stoptelescope();
	command_timeout(IN := TCS_command = E_TCSCommand.stop, PT := T#2S);
	TCSCTOEvent.OnMessage := 'STOP';
ELSIF TCS_command = E_TCSCommand.park THEN
	parktelescope();
	command_timeout(IN := TCS_command = E_TCSCommand.park, PT := T#2M);
	TCSCTOEvent.OnMessage := 'PARK';
ELSIF TCS_command = E_TCSCommand.gohome THEN
	hometelescope();
	command_timeout(IN := TCS_command = E_TCSCommand.gohome, PT := T#2M);
	TCSCTOEvent.OnMessage := 'GOHOME';
ELSIF TCS_command = E_TCSCommand.goto THEN
	gototelescope();
	command_timeout(IN := TCS_command = E_TCSCommand.goto, PT := T#2M);
	TCSCTOEvent.OnMessage := 'GOTO';
ELSIF TCS_command = E_TCSCommand.slew THEN
	slewtelescope();
	command_timeout(IN := TCS_command = E_TCSCommand.slew, PT := T#2M);
	TCSCTOEvent.OnMessage := 'SLEW';
ELSIF TCS_command = E_TCSCommand.track THEN
	tracktelescope();
	command_timeout(IN := TCS_command = E_TCSCommand.track, PT := T#12H);
	TCSCTOEvent.OnMessage := 'TRACK';
ELSE
	// disable command timeout
	command_timeout(IN := FALSE);
	TCSCTOEvent.OnMessage := 'NOCOMMAND';
END_IF
 
sliding := NOT tracking AND (ElevationControl.ElevationAxis.InMotion OR ElevationControl.ElevationAxis.InRamp OR
			AzimuthElevationControl.AzimuthAxis.InMotion OR AzimuthElevationControl.AzimuthAxis.InRamp OR
			DerotatorControl.DerotatorAxis.InMotion OR DerotatorControl.DerotatorAxis.InRamp);

// signal must be stable for 5500MS
tracking_delay(in := ElevationControl.ElevationAxis.isTracking AND 
			AzimuthElevationControl.AzimuthAxis.isTracking AND
			DerotatorControl.DerotatorAxis.isTracking,PT :=T#5500MS, Q => tracking);
			
stopped :=  (NOT ElevationControl.enable OR ElevationControl.ElevationAxis.StandStill) AND 
			(NOT AzimuthElevationControl.Enable OR AzimuthElevationControl.AzimuthAxis.StandStill) AND
			(NOT DerotatorControl.enable OR DerotatorControl.DerotatorAxis.StandStill);
			
homed := ElevationControl.Calibrated AND
			AzimuthElevationControl.calibrated AND
			FocusControl.Calibrated AND
			DerotatorControl.Calibrated;
			
ready := homed AND 
	CoverControl.isopen AND 
	ElevationControl.enable AND
	AzimuthElevationControl.enable AND
	DerotatorControl.enable AND HydraulicsControl.brake_open AND 
    NOT error;

busy := ElevationControl.ElevationAxis.Busy OR
		AzimuthElevationControl.AzimuthAxis.Busy OR
		DerotatorControl.DerotatorAxis.Busy OR
		FocusControl.FocusAxis.Busy;

// unset the STOP command if telescope is already stopped
IF stopped THEN
	stop := FALSE;
END_IF
	
IF NOT error THEN
	reset := FALSE;
END_IF

IF SafetyHandling.Emergency_stop THEN
	ElevationControl.enable := FALSE;
	AzimuthElevationControl.enable := FALSE;
	DerotatorControl.enable := FALSE;
END_IF
IF sliding OR track OR tracking THEN
	MQTTTimer.PT := T#1000MS;
ELSE
	MQTTTimer.PT := T#5000MS;
END_IF
MQTTTimer(IN:=TRUE);
IF MQTTTimer.Q THEN // publish new payload every second
	MQTTTimer(IN:=FALSE);

	MAIN.MQTTClient.Publish('telescope', 'dome', 'JulianDate', LREAL_TO_STRING(jd));
	MAIN.MQTTClient.Publish('telescope', 'dome', 'LocalSiderialTime', LREAL_TO_STRING(lst));
	MAIN.MQTTClient.Publish('telescope', 'dome', 'Azimuth', LREAL_TO_STRING(azimuth_current));
	MAIN.MQTTClient.Publish('telescope', 'dome', 'Elevation', LREAL_TO_STRING(elevation_current));
	MAIN.MQTTClient.Publish('telescope', 'dome', 'Derotator', LREAL_TO_STRING(derotator_current));
	MAIN.MQTTClient.Publish('telescope', 'dome', 'HourAngle', LREAL_TO_STRING(hourangle_calc));
	MAIN.MQTTClient.Publish('telescope', 'dome', 'RightAscension', LREAL_TO_STRING(rightascension_calc));
	MAIN.MQTTClient.Publish('telescope', 'dome', 'Declination', LREAL_TO_STRING(declination_calc));
	MAIN.MQTTClient.Publish('telescope', 'dome', 'azimuth_offset', LREAL_TO_STRING(azimuth_offset));
	MAIN.MQTTClient.Publish('telescope', 'dome', 'elevation_offset', LREAL_TO_STRING(elevation_offset));
	MAIN.MQTTClient.Publish('telescope', 'dome', 'derotator_torque', LREAL_TO_STRING(DerotatorControl.derotator_torque));
	MAIN.MQTTClient.Publish('telescope', 'dome', 'elevation_torque', LREAL_TO_STRING(ElevationControl.elevation_torque));
	MAIN.MQTTClient.Publish('telescope', 'dome', 'azimuth_torque', LREAL_TO_STRING(AzimuthElevationControl.azimuth_torque));
	
	MAIN.MQTTClient.Publish('telescope', 'dome', 'errorid',		UDINT_TO_STRING(errorid));
	MAIN.MQTTClient.Publish('telescope', 'dome', 'error',		BOOL_TO_STRING(error));
	MAIN.MQTTClient.Publish('telescope', 'dome', 'ready',		BOOL_TO_STRING(ready));
	MAIN.MQTTClient.Publish('telescope', 'dome', 'busy',		BOOL_TO_STRING(busy));
	MAIN.MQTTClient.Publish('telescope', 'dome', 'sliding',		BOOL_TO_STRING(sliding));
	MAIN.MQTTClient.Publish('telescope', 'dome', 'tracking', 	BOOL_TO_STRING(tracking));
	MAIN.MQTTClient.Publish('telescope', 'dome', 'stopped',		BOOL_TO_STRING(stopped));
	MAIN.MQTTClient.Publish('telescope', 'dome', 'homed',		BOOL_TO_STRING(homed));
END_IF

StatusWord.0 := error;
StatusWord.1 := ready;
StatusWord.2 := sliding;
StatusWord.3 := tracking;
StatusWord.4 := stopped;
StatusWord.5 := homed;
StatusWord.6 := power;
StatusWord.7 := park;
StatusWord.8 := gohome;
StatusWord.9 := track;
StatusWord.10 := goto;
StatusWord.11 := slew;
StatusWord.12 := stop;
StatusWord.13 := busy;

IF StatusWord<>LastStatus THEN // publish new payload every second
	LastStatus := StatusWord;
	MAIN.MQTTClient.Publish('telescope', 'dome', 'error',		BOOL_TO_STRING(error));
	MAIN.MQTTClient.Publish('telescope', 'dome', 'ready',		BOOL_TO_STRING(ready));
	MAIN.MQTTClient.Publish('telescope', 'dome', 'sliding',		BOOL_TO_STRING(sliding));
	MAIN.MQTTClient.Publish('telescope', 'dome', 'tracking', 	BOOL_TO_STRING(tracking));
	MAIN.MQTTClient.Publish('telescope', 'dome', 'stopped',		BOOL_TO_STRING(stopped));
	MAIN.MQTTClient.Publish('telescope', 'dome', 'homed',		BOOL_TO_STRING(homed));
	MAIN.MQTTClient.Publish('telescope', 'dome', 'power',		BOOL_TO_STRING(power));
	MAIN.MQTTClient.Publish('telescope', 'dome', 'park',		BOOL_TO_STRING(park));
	MAIN.MQTTClient.Publish('telescope', 'dome', 'gohome',		BOOL_TO_STRING(gohome));
	MAIN.MQTTClient.Publish('telescope', 'dome', 'track',		BOOL_TO_STRING(track));
	MAIN.MQTTClient.Publish('telescope', 'dome', 'goto',		BOOL_TO_STRING(goto));
	MAIN.MQTTClient.Publish('telescope', 'dome', 'slew',		BOOL_TO_STRING(slew));
	MAIN.MQTTClient.Publish('telescope', 'dome', 'stop',		BOOL_TO_STRING(stop));
	MAIN.MQTTClient.Publish('telescope', 'dome', 'busy',		BOOL_TO_STRING(busy));
END_IF


(* Event function blocks start here. *)
TCSpowerEvent(	Trigger := powerfailure, 
				Level := ADSLOG_MSGTYPE_ERROR,
				FormatString := 'power %s',
				OnMessage := 'Failure',
				OffMessage := 'OK');

TCSgohomeEvent(	Trigger := gohome, 
				Level := ADSLOG_MSGTYPE_HINT,
				FormatString := 'GOHOME %s',
				OnMessage := 'commencing',
				OffMEssage := 'completed');
TCSparkEvent(	Trigger := park, 
				Level := ADSLOG_MSGTYPE_HINT,
				FormatString := 'PARK %s',
				OnMessage := 'commencing',
				OffMEssage := 'completed');
TCSgotoEvent(	Trigger := goto, 
				Level := ADSLOG_MSGTYPE_HINT,
				FormatString := 'GOTO %s',
				OnMessage := 'commencing',
				OffMEssage := 'completed');
TCStrackEvent(	Trigger := track, 
				Level := ADSLOG_MSGTYPE_HINT,
				FormatString := 'TRACK %s',
				OnMessage := 'commencing',
				OffMEssage := 'completed');
TCSstopEvent(	Trigger := stop, 
				Level := ADSLOG_MSGTYPE_WARN,
				FormatString := 'STOP %s',
				OnMessage := 'commencing',
				OffMEssage := 'completed',
				OffLevel := ADSLOG_MSGTYPE_HINT);
AltitudeEvent(	Trigger := power AND elevation_calc<0.0, 
				Level := ADSLOG_MSGTYPE_WARN,
				FormatString := '%s',
				OnMessage := 'Target below horizon',
				OffMEssage := '');
TCSreadyEvent(	Trigger := power AND ready, 
				Level := ADSLOG_MSGTYPE_HINT,
				FormatString := '%s',
				OnMessage := 'STELLA1 startup finished');
TCSCTOEvent(	Trigger := command_timeout.Q,
				Level := ADSLOG_MSGTYPE_WARN,
				FormatString := 'A timeout occured during %s command!',
				OnMessage := 'NOCOMMAND');

METHOD gototelescope: USINT
VAR_INPUT
END_VAR
VAR
	GoToEvent:	FB_Eventlog;
	command_timeout:	TON;
END_VAR
VAR_STAT
	Stage:		USINT := 0;
	LastStage:	USINT := 101;
END_VAR
gototelescope := Stage;
command_timeout(IN := Stage < 100, PT := T#600S);
IF command_timeout.Q THEN
	error := TRUE;
	errorid := 16#10;
	goto := FALSE;
	Stage := 0;
	RETURN;
END_IF

IF elevation_calc<2.0 THEN
	error := TRUE;
	errorid := 16#15;
	goto := FALSE;
	Stage := 0;
	RETURN;
END_IF

IF reset OR error THEN
	Stage := 0;
	RETURN;
END_IF

CASE Stage OF
	0:	
		IF ready AND NOT busy THEN
			Stage := 25;
		END_IF
	25:	
		ElevationControl.position := elevation_calc;
		AzimuthElevationControl.position := azimuth_calc;
		DerotatorControl.position := derotation_calc;
		DerotatorControl.Velocity := 10.0;
		ElevationControl.velocity := 10.0;
		AzimuthElevationControl.velocity := 10.0;
		
		ElevationControl.MoveAxis := TRUE;
		AzimuthElevationControl.MoveAxis := TRUE;
		DerotatorControl.MoveAxis := TRUE;
		IF ElevationControl.ElevationAxis.Busy AND
			AzimuthElevationControl.AzimuthAxis.Busy AND
			DerotatorControl.DerotatorAxis.Busy THEN
				Stage := 50;
		END_IF
	50:
		IF NOT ElevationControl.ElevationAxis.Busy AND ElevationControl.ElevationAxis.MoveDone THEN
			ElevationControl.MoveAxis := FALSE;
		END_IF
		IF NOT AzimuthElevationControl.AzimuthAxis.Busy AND AzimuthElevationControl.AzimuthAxis.MoveDone THEN
			AzimuthElevationControl.MoveAxis := FALSE;
		END_IF
		IF NOT DerotatorControl.DerotatorAxis.Busy AND DerotatorControl.DerotatorAxis.MoveDone THEN
			DerotatorControl.MoveAxis := FALSE;
		END_IF
		IF NOT ElevationControl.MoveAxis AND 
           NOT AzimuthElevationControl.MoveAxis AND 
		   NOT DerotatorControl.MoveAxis THEN
		   Stage := 75;
		END_IF
	75:
		IF NOT sliding AND stopped THEN // all axis standstill
			Stage := 100;
		END_IF
	100:
		ElevationControl.MoveAxis := FALSE;
		AzimuthElevationControl.MoveAxis := FALSE;
		DerotatorControl.MoveAxis := FALSE;
		azimuth := azimuth_calc;
		elevation := elevation_calc;
		goto := FALSE;
		// enable automatic tracking
		track := autotrack;
		Stage := 0;
END_CASE
GoToEvent(Trigger := Stage > LastStage, FormatString := 'GoTo progress: %s', OnMessage := USINT_TO_STRING(Stage));
LastStage := Stage;
END_METHOD

METHOD hometelescope : BOOL
VAR_INPUT
END_VAR

VAR
	HomeEvent: FB_Eventlog;
	command_timeout: TON;
END_VAR
command_timeout(IN := NOT hometelescope, PT := T#600S);
IF command_timeout.Q THEN
	error := TRUE;
	errorid := 16#30;
	hometelescope :=TRUE;
END_IF

IF ready AND stopped AND NOT busy AND NOT tracking THEN
	ElevationControl.velocity := 10.0;
	ElevationControl.position := elevation_home;
	ElevationControl.MoveAxis := TRUE;
	AzimuthElevationControl.velocity := 10.0;
	AzimuthElevationControl.position := azimuth_home;
	AzimuthElevationControl.MoveAxis := TRUE;
	DerotatorControl.Velocity := 10.0;
	DerotatorControl.position := 180.0;
	DerotatorControl.MoveAxis := TRUE;	
END_IF

IF ElevationControl.ElevationAxis.MoveDone AND 
	AzimuthElevationControl.AzimuthAxis.MoveDone AND 
	DerotatorControl.DerotatorAxis.MoveDone THEN
	gohome := FALSE;
	elevation := elevation_current;
	azimuth := azimuth_current;
	hometelescope := TRUE;
ELSE
	hometelescope := FALSE;
END_IF

HomeEvent(Trigger := hometelescope, 
			Level := ADSLOG_MSGTYPE_HINT,
			FormatString := '%s',
			OnMessage := 'Telescope is homed.');
END_METHOD

METHOD parktelescope: USINT
VAR_INPUT
END_VAR
VAR
	ParkEvent:	FB_Eventlog;
END_VAR
VAR_STAT
	Stage:		USINT := 0;
	LastStage:	USINT := 101;
END_VAR
parktelescope := Stage;
IF reset OR error THEN
	Stage := 0;
END_IF
IF isparked THEN
	Stage := 100;
END_IF
CASE Stage OF
	0: 
		gohome := 	FALSE;
		track := 	FALSE;
		goto := 	FALSE;
		slew := 	FALSE;
		Focuscontrol.position := 53.6;
		IF Error THEN // emergency park
			HydraulicsControl.close_brake();
			ElevationControl.enable := FALSE;
			AzimuthElevationControl.Enable := FALSE;
			DerotatorControl.enable := FALSE;	
			CoverControl.close := TRUE;	
			Stage := 80;
		END_IF
		Stage := 20;
	20:
		ElevationControl.position := elevation_park;
		ElevationControl.velocity := 10.0;
		ElevationControl.MoveAxis := TRUE;
		AzimuthElevationControl.position := azimuth_park;
		AzimuthElevationControl.velocity := 10;
		AzimuthElevationControl.MoveAxis := TRUE;
		DerotatorControl.position := derotator_park;
		DerotatorControl.Velocity := 10.0;
		DerotatorControl.MoveAxis := TRUE;
		IF ElevationControl.ElevationAxis.Busy AND
			AzimuthElevationControl.AzimuthAxis.Busy AND
			DerotatorControl.DerotatorAxis.Busy THEN
				Stage := 40;
		END_IF
	40:
		IF ElevationControl.ElevationAxis.MoveDone THEN
			ElevationControl.MoveAxis := FALSE;
		END_IF
		IF AzimuthElevationControl.AzimuthAxis.MoveDone THEN
			AzimuthElevationControl.MoveAxis := FALSE;
		END_IF
		IF DerotatorControl.DerotatorAxis.MoveDone THEN
			DerotatorControl.MoveAxis := FALSE;
		END_IF
		IF NOT sliding THEN // all axis standstill
			Stage := 60;
		END_IF
	60:
		IF NOT ElevationControl.enable AND NOT AzimuthElevationControl.Enable AND NOT DerotatorControl.enable THEN
			stage := 80;
		END_IF

		IF stopped THEN
			ElevationControl.enable := FALSE;
			AzimuthElevationControl.Enable := FALSE;
			DerotatorControl.enable := FALSE;
		END_IF
		
		ElevationControl.MoveAxis := FALSE;
		AzimuthElevationControl.MoveAxis := FALSE;
		DerotatorControl.MoveAxis := FALSE;
	80:
		IF ElevationControl.enable OR AzimuthElevationControl.Enable OR DerotatorControl.enable THEN
			stage := 60;
		END_IF
		IF HydraulicsControl.brake_closed THEN
			CoverControl.close := TRUE;
			HydraulicsControl.enable := FALSE;
		END_IF
		IF CoverControl.isclosed THEN
			Stage := 100;
		END_IF
	100:
			isparked := TRUE;
			park := FALSE;
			parktelescope := 100;
			Stage := 0;	
END_CASE
ParkEvent(Trigger := Stage > LastStage, FormatString := 'Parking progress: %s', OnMessage := USINT_TO_STRING(Stage));
LastStage := Stage;
END_METHOD

METHOD poweron : BOOL
VAR_INPUT
END_VAR
VAR
END_VAR
IF NOT Main.brake_clearing THEN
	powerfailure := TRUE;
	TCSpowerEvent.OnMessage := 'failure: brake clearing not set';
	power := FALSE;
ELSIF error THEN
	powerfailure := TRUE;
	TCSpowerEvent.OnMessage := 'Generic error during power on occured.';
	power := FALSE;
ELSE
	powerfailure := FALSE;		
END_IF
// COVER MUST BE OPENED FOR A SUCCESSFUL WAKE & SHAKE COMMAND!
Covercontrol.open := TRUE;

// enable elevation, enable azimuth
IF MAIN.ready AND CoverControl.isopen THEN
	ElevationControl.enable := TRUE;
	AzimuthElevationControl.enable := TRUE;
	DerotatorControl.enable := TRUE;
END_IF

IF ElevationControl.Ready AND NOT ElevationControl.Calibrated THEN
	ElevationControl.HomeAxis := TRUE;
END_IF

IF AzimuthElevationControl.ready AND NOT AzimuthElevationControl.calibrated THEN
	AzimuthElevationControl.HomeAxis := TRUE;
END_IF

// enable derotator
IF ElevationControl.Ready THEN
	DerotatorControl.HomeAxis := DerotatorControl.Ready AND NOT DerotatorControl.Calibrated;
END_IF

// start calibration of focus after elevation has been calibrated
// this avoids imbalance by the M2 mirror on the elvation during its calibration
IF ElevationControl.Calibrated AND NOT FocusControl.Calibrated THEN
	FocusControl.enable := TRUE;
	FocusControl.HomeAxis := TRUE;
END_IF

IF CoverControl.isopen AND 
	ElevationControl.Calibrated AND
	AzimuthElevationControl.calibrated AND
	DerotatorControl.Calibrated AND
	FocusControl.Calibrated THEN
	power := FALSE;
	poweron := TRUE;
	isparked := FALSE;
	// slew the telescope to the home position
	gohome := TRUE;
ELSE
	poweron := FALSE;
END_IF
END_METHOD

METHOD slewtelescope : USINT
VAR_INPUT
END_VAR
VAR
	SlewEvent:	FB_Eventlog;
	command_timeout: TON;
END_VAR
VAR_STAT
	Stage:		USINT := 0;
	LastStage:	USINT := 101;
END_VAR
slewtelescope := Stage;
command_timeout(IN := Stage < 100, PT := T#600S);
IF command_timeout.Q THEN
	error := TRUE;
	errorid := 16#40;
	slew := FALSE;
	Stage := 0;
END_IF
IF reset OR error THEN
	Stage := 0;
END_IF
CASE Stage OF
	0:	
		IF ready AND stopped AND NOT busy AND NOT tracking THEN
			Stage := 25;
		END_IF
	25:
		ElevationControl.position := elevation;
		ElevationControl.velocity := 10.0;
		ElevationControl.MoveAxis := TRUE;
		AzimuthElevationControl.position := azimuth;
		AzimuthElevationControl.velocity := 10.0;
		AzimuthElevationControl.MoveAxis := TRUE;
		DerotatorControl.position := elevation + derotator_offset;
		DerotatorControl.Velocity := 10.0;
		DerotatorControl.MoveAxis := TRUE;
		IF ElevationControl.ElevationAxis.Busy AND
			AzimuthElevationControl.AzimuthAxis.Busy AND
			DerotatorControl.DerotatorAxis.Busy THEN
				Stage := 50;
		END_IF
	50:
		IF ElevationControl.ElevationAxis.MoveDone THEN
			ElevationControl.MoveAxis := FALSE;
		END_IF
		
		IF AzimuthElevationControl.AzimuthAxis.MoveDone THEN
			AzimuthElevationControl.MoveAxis := FALSE;
		END_IF

		IF DerotatorControl.DerotatorAxis.MoveDone THEN
			DerotatorControl.MoveAxis := FALSE;
		END_IF
		IF NOT sliding AND stopped THEN // all axis standstill
			Stage := 100;
		END_IF
	100:
		ElevationControl.MoveAxis := FALSE;
		AzimuthElevationControl.MoveAxis := FALSE;
		DerotatorControl.MoveAxis := FALSE;
		rightascension := rightascension_calc;
		declination := declination_calc;
		slew := FALSE;
		Stage := 0;
END_CASE
SlewEvent(Trigger := Stage > LastStage, FormatString := 'Slew progress: %s', OnMessage := USINT_TO_STRING(Stage));
LastStage := Stage;
END_METHOD

METHOD stoptelescope : BOOL
VAR_INPUT
END_VAR
ElevationControl.StopAxis := TRUE;
AzimuthElevationControl.StopAxis := TRUE;
DerotatorControl.StopAxis := TRUE;
IF stopped THEN
	ElevationControl.StopAxis := FALSE;
	AzimuthElevationControl.StopAxis := FALSE;
	DerotatorControl.StopAxis := FALSE;
	stop := FALSE;
END_IF
END_METHOD

METHOD tracktelescope : BOOL
VAR_INPUT
END_VAR
// Elevation
DerotatorVelocity := F_Derotatorvelocity(elevation_calc, azimuth_calc, latitude);
ElevationVelocity := F_Elevationvelocity(azimuth_calc, latitude);
AzimuthVelocity := F_Azimuthvelocity(elevation_calc, azimuth_calc, latitude);
IF elevation_current < 5.0 OR elevation_current > 89.5 THEN 
	track := FALSE;
END_IF
IF azimuth_current > 440.0 THEN
	track := FALSE;
END_IF
IF (derotator_current < -69.0 AND DerotatorVelocity<0.0) OR (derotator_current > 379.0 AND DerotatorVelocity>0.0) THEN
	track := FALSE;
END_IF

ElevationControl.position := elevation_calc;
IF NOT ElevationControl.Tracking THEN
	ElevationControl.velocity := 10.0;
	ElevationControl.MoveAxis := TRUE;
	IF NOT ElevationControl.ElevationAxis.Busy AND ElevationControl.ElevationAxis.MoveDone THEN
		ElevationControl.MoveAxis := FALSE;
		IF ElevationControl.ElevationAxis.isTracking THEN
			ElevationControl.velocity := ElevationVelocity;
		ELSE
			ElevationControl.velocity := 3.0*ElevationVelocity;
		END_IF
		ElevationControl.velocity := ElevationVelocity;
		ElevationControl.Tracking := TRUE;
	END_IF
ELSE
	ElevationControl.velocity := ElevationVelocity;
END_IF

// Azimuth
AzimuthElevationControl.position := azimuth_calc;
IF NOT AzimuthElevationControl.Tracking THEN
	AzimuthElevationControl.velocity := 10.0;
	AzimuthElevationControl.MoveAxis := TRUE;
	IF NOT AzimuthElevationControl.AzimuthAxis.Busy AND AzimuthElevationControl.AzimuthAxis.MoveDone THEN
		AzimuthElevationControl.MoveAxis := FALSE;
		IF AzimuthElevationControl.AzimuthAxis.isTracking THEN
			AzimuthElevationControl.velocity := AzimuthVelocity;
		ELSE
			AzimuthElevationControl.velocity := 3.0*AzimuthVelocity;
		END_IF
		AzimuthElevationControl.velocity := AzimuthVelocity;
		AzimuthElevationControl.Tracking := TRUE;
	END_IF
ELSE
	AzimuthElevationControl.velocity := AzimuthVelocity;
END_IF

// Derotator
DerotatorControl.position := derotation_calc;
IF NOT DerotatorControl.Tracking THEN
	DerotatorControl.Velocity := 10.0;
	DerotatorControl.MoveAxis := TRUE;
	IF NOT DerotatorControl.DerotatorAxis.Busy AND DerotatorControl.DerotatorAxis.MoveDone THEN
		DerotatorControl.MoveAxis := FALSE;
		IF DerotatorControl.DerotatorAxis.isTracking THEN
			DerotatorControl.Velocity := DerotatorVelocity;
		ELSE
			DerotatorControl.Velocity := 3.0*DerotatorVelocity;
		END_IF
		DerotatorControl.Velocity := DerotatorVelocity;
		DerotatorControl.Tracking := TRUE;
	END_IF
ELSE
	DerotatorControl.Velocity := DerotatorVelocity;
END_IF
END_METHOD

END_PROGRAM

// ---- POUs/TelescopeAuxiliary.TcPOU
PROGRAM TelescopeAuxiliary
VAR
	MQTTTimer : TON := (PT:=T#5S);
END_VAR
VAR_INPUT
	comm: I_Comm;
END_VAR
VAR_OUTPUT
	// BT9 mirror
	temperature_mirror2:	REAL;
	// BT10
	temperature_mirror1:	REAL;
END_VAR

//temperature_mirror1 := GVL_Telescope.temperature_mirror1 / 1000.0;
//temperature_mirror2 := GVL_Telescope.temperature_mirror2 / 1000.0;
temperature_mirror1 := GVL_Telescope.temperature_mirror1 / 32767.0 * 150.0 - 50.0;
temperature_mirror2 := GVL_Telescope.temperature_mirror2 / 32767.0 * 150.0 - 50.0;

MQTTTimer(IN:=TRUE);
IF MQTTTimer.Q THEN // publish new payload every second

